KUKA KRL program: EPS_2_25369_MH3A_A_20251215023756.src

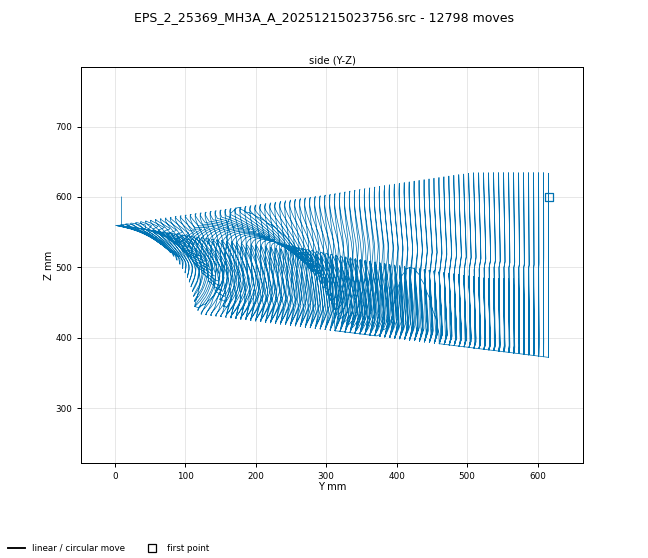
[picture p0: tool path of EPS_2_25369_MH3A_A_20251215023756.src, 12798 of 12800 moves have a stored position in this frame; points joined in program order, loops and branches not executed]
&ACCESS RVP
&REL 4
&COMMENT QRS 19112012
&PARAM EDITMASK = *
DEF PART()
EXT BAS (BAS_COMMAND :IN,REAL :IN )
INT I
BAS (#INITMOV,0 )

;KUKA QRS Post kuka4.cps  Date:22-06-2017 !

File_ID=2956

QRS_PRE_INIT()

;Init var - Until changes are made in qrs_pre_init
Outlet_Square_prg=0
Inlet_1_Square_prg=0
Inlet_2_Square_prg=0
Inlet_3_Square_prg=0
Inlet_4_Square_prg=0
Inlet_5_Square_prg=0

Outlet_1={X 0.000, Y 509.470, Z 509.000, B 0.000, E1 0.000 }
Inlet_1={X 0.000, Y 526.260, Z 384.000, B 0.000, E1 183.000 }
Inlet_2={X 0.000, Y 520.510, Z 359.000, B 0.000, E1 271.000 }
Outlet_1_type=251
Inlet_1_type=201
Inlet_2_type=251
;QRS#1=Sidecore dimensions
;QRS#2=250-10" PVC SDR 35
;QRS#3=200-8" PVC SDR 35
;QRS#4=250-10" PVC SDR 35
;QRS#5=
;QRS#6=
;QRS#7=
;QRS#8=
;QRS#9=14M PSX
;QRS#10=12-08 PSX
;QRS#11=14M PSX
;QRS#12=
;QRS#13=
;QRS#14=
;QRS#15=
;QRS#16=1220x127x914 3'
;QRS#17=EPS Height
;QRS#18=634,5
;QRS#19=*
;QRS#20= UPDATED VERSION 22-06-2017
;QRS#21=*
Outlet_Square=0100
Inlet_1_Square=0100
Inlet_2_Square=0100
Inlet_3_Square=0
Inlet_4_Square=0
Inlet_5_Square=0
Mill_Square=1
Outlet_Square_Prg=205
Inlet_1_Square_prg=204
Inlet_2_Square_prg=205

QRS_INIT()

$ADVANCE=5

; T1
PTP {E1 173.595,E2 173.595}
PTP {X 0,Y 615.506,A -85,B 0,C 180,E1 173.595,E2 173.595,E3 0,E4 0,E5 0,E6 0}
QRS_SPEED_INIT()
LIN {X 0,Y 615.506,Z 600,A -85,B 0,C 180,E1 173.595,E2 173.595,E3 0,E4 0,E5 0,E6 0} C_VEL
LIN {X 0,Y 615.506,Z 382.487,A -85,B 0,C 180,E1 173.595,E2 173.595} C_VEL
LIN {X 0,Y 615.506,Z 374.307,A -85,B 0,C 180,E1 173.595,E2 173.595} C_VEL
LIN {X 0,Y 615.49,Z 372.307,A -85,B 0,C 180,E1 173.408,E2 173.408} C_VEL
LIN {X 0,Y 615.486,Z 372.321,A -85,B 0,C 180,E1 170.801,E2 170.801} C_VEL
LIN {X 0,Y 615.474,Z 372.316,A -85,B 0,C 180,E1 168.139,E2 168.139} C_VEL
LIN {X 0,Y 615.49,Z 372.307,A -85,B 0,C 180,E1 165.451,E2 165.451} C_VEL
LIN {X 0,Y 615.494,Z 372.324,A -85,B 0,C 180,E1 162.729,E2 162.729} C_VEL
LIN {X 0,Y 615.479,Z 372.311,A -85,B 0,C 180,E1 159.967,E2 159.967} C_VEL
LIN {X 0,Y 615.491,Z 372.306,A -85,B 0,C 180,E1 157.65,E2 157.65} C_VEL
LIN {X 0,Y 615.48,Z 372.319,A -85,B 0,C 180,E1 155.008,E2 155.008} C_VEL
LIN {X 0,Y 615.487,Z 372.324,A -85,B 0,C 180,E1 152.822,E2 152.822} C_VEL
LIN {X 0,Y 615.477,Z 372.314,A -85,B 0,C 180,E1 150.205,E2 150.205} C_VEL
LIN {X 0,Y 615.49,Z 372.307,A -85,B 0,C 180,E1 147.542,E2 147.542} C_VEL
LIN {X 0,Y 615.481,Z 372.316,A -85,B 0,C 180,E1 145.184,E2 145.184} C_VEL
LIN {X 0,Y 615.494,Z 372.325,A -85,B 0,C 180,E1 142.758,E2 142.758} C_VEL
LIN {X 0,Y 615.486,Z 372.307,A -85,B 0,C 180,E1 139.909,E2 139.909} C_VEL
LIN {X 0,Y 615.494,Z 372.306,A -85,B 0,C 180,E1 137.647,E2 137.647} C_VEL
LIN {X 0,Y 615.491,Z 372.324,A -85,B 0,C 180,E1 134.931,E2 134.931} C_VEL
LIN {X 0,Y 615.48,Z 372.31,A -85,B 0,C 180,E1 132.079,E2 132.079} C_VEL
LIN {X 0,Y 615.494,Z 372.306,A -85,B 0,C 180,E1 129.748,E2 129.748} C_VEL
LIN {X 0,Y 615.488,Z 372.327,A -85,B 0,C 180,E1 126.936,E2 126.936} C_VEL
LIN {X 0,Y 615.491,Z 372.319,A -85,B 0,C 180,E1 124.7,E2 124.7} C_VEL
LIN {X 0,Y 615.477,Z 372.312,A -85,B 0,C 180,E1 122.328,E2 122.328} C_VEL
LIN {X 0,Y 615.497,Z 372.305,A -85,B 0,C 180,E1 119.795,E2 119.795} C_VEL
LIN {X 0,Y 615.491,Z 372.325,A -85,B 0,C 180,E1 117.045,E2 117.045} C_VEL
LIN {X 0,Y 615.478,Z 372.311,A -85,B 0,C 180,E1 114.271,E2 114.271} C_VEL
LIN {X 0,Y 615.481,Z 372.316,A -85,B 0,C 180,E1 111.431,E2 111.431} C_VEL
LIN {X 0,Y 615.481,Z 372.315,A -85,B 0,C 180,E1 108.602,E2 108.602} C_VEL
LIN {X 0,Y 615.487,Z 372.308,A -85,B 0,C 180,E1 105.904,E2 105.904} C_VEL
LIN {X 0,Y 615.49,Z 372.321,A -85,B 0,C 180,E1 105.225,E2 105.225} C_VEL
LIN {X 0,Y 615.478,Z 375.734,A -85,B 0,C 180,E1 102.529,E2 102.529} C_VEL
LIN {X 0,Y 615.491,Z 379.183,A -85,B 0,C 180,E1 99.861,E2 99.861} C_VEL
LIN {X 0,Y 615.482,Z 380.919,A -85,B 0,C 180,E1 98.536,E2 98.536} C_VEL
LIN {X 0,Y 615.488,Z 393.813,A -85,B 0,C 180,E1 98.246,E2 98.246} C_VEL
LIN {X 0,Y 615.485,Z 406.345,A -85,B 0,C 180,E1 97.834,E2 97.834} C_VEL
LIN {X 0,Y 615.478,Z 418.326,A -85,B 0,C 180,E1 97.297,E2 97.297} C_VEL
LIN {X 0,Y 615.495,Z 429.344,A -85,B 0,C 180,E1 96.661,E2 96.661} C_VEL
LIN {X 0,Y 615.5,Z 439.937,A -85,B 0,C 180,E1 95.898,E2 95.898} C_VEL
LIN {X 0,Y 615.498,Z 449.187,A -85,B 0,C 180,E1 95.076,E2 95.076} C_VEL
LIN {X 0,Y 615.499,Z 458.111,A -85,B 0,C 180,E1 94.092,E2 94.092} C_VEL
LIN {X 0,Y 615.497,Z 465.316,A -85,B 0,C 180,E1 93.108,E2 93.108} C_VEL
LIN {X 0,Y 615.5,Z 471.91,A -85,B 0,C 180,E1 91.962,E2 91.962} C_VEL
LIN {X 0,Y 615.497,Z 476.278,A -85,B 0,C 180,E1 90.981,E2 90.981} C_VEL
LIN {X 0,Y 615.496,Z 479.593,A -85,B 0,C 180,E1 89.999,E2 89.999} C_VEL
LIN {X 0,Y 615.498,Z 482.486,A -85,B 0,C 180,E1 88.691,E2 88.691} C_VEL
LIN {X 0,Y 615.499,Z 483.348,A -85,B 0,C 180,E1 88.036,E2 88.036} C_VEL
LIN {X 0,Y 615.496,Z 483.794,A -85,B 0,C 180,E1 87.381,E2 87.381} C_VEL
LIN {X 0,Y 615.495,Z 483.512,A -85,B 0,C 180,E1 86.071,E2 86.071} C_VEL
LIN {X 0,Y 615.496,Z 482.804,A -85,B 0,C 180,E1 85.415,E2 85.415} C_VEL
LIN {X 0,Y 615.496,Z 481.658,A -85,B 0,C 180,E1 84.758,E2 84.758} C_VEL
LIN {X 0,Y 615.497,Z 480.101,A -85,B 0,C 180,E1 84.101,E2 84.101} C_VEL
LIN {X 0,Y 615.497,Z 476.921,A -85,B 0,C 180,E1 83.101,E2 83.101} C_VEL
LIN {X 0,Y 615.495,Z 472.771,A -85,B 0,C 180,E1 82.124,E2 82.124} C_VEL
LIN {X 0,Y 615.496,Z 466.374,A -85,B 0,C 180,E1 80.966,E2 80.966} C_VEL
LIN {X 0,Y 615.497,Z 459.364,A -85,B 0,C 180,E1 79.971,E2 79.971} C_VEL
LIN {X 0,Y 615.498,Z 450.403,A -85,B 0,C 180,E1 78.958,E2 78.958} C_VEL
LIN {X 0,Y 615.497,Z 441.497,A -85,B 0,C 180,E1 78.139,E2 78.139} C_VEL
LIN {X 0,Y 615.5,Z 431.437,A -85,B 0,C 180,E1 77.386,E2 77.386} C_VEL
LIN {X 0,Y 615.477,Z 420.231,A -85,B 0,C 180,E1 76.714,E2 76.714} C_VEL
LIN {X 0,Y 615.487,Z 409.605,A -85,B 0,C 180,E1 76.209,E2 76.209} C_VEL
LIN {X 0,Y 615.491,Z 397.137,A -85,B 0,C 180,E1 75.758,E2 75.758} C_VEL
LIN {X 0,Y 615.484,Z 383.804,A -85,B 0,C 180,E1 75.429,E2 75.429} C_VEL
LIN {X 0,Y 615.484,Z 380.908,A -85,B 0,C 180,E1 75.366,E2 75.366} C_VEL
LIN {X 0,Y 615.477,Z 377.471,A -85,B 0,C 180,E1 72.729,E2 72.729} C_VEL
LIN {X 0,Y 615.486,Z 373.927,A -85,B 0,C 180,E1 69.967,E2 69.967} C_VEL
LIN {X 0,Y 615.487,Z 372.319,A -85,B 0,C 180,E1 68.568,E2 68.568} C_VEL
LIN {X 0,Y 615.478,Z 372.311,A -85,B 0,C 180,E1 65.727,E2 65.727} C_VEL
LIN {X 0,Y 615.491,Z 372.324,A -85,B 0,C 180,E1 62.955,E2 62.955} C_VEL
LIN {X 0,Y 615.497,Z 372.306,A -85,B 0,C 180,E1 60.205,E2 60.205} C_VEL
LIN {X 0,Y 615.481,Z 372.318,A -85,B 0,C 180,E1 57.542,E2 57.542} C_VEL
LIN {X 0,Y 615.499,Z 372.322,A -85,B 0,C 180,E1 55.185,E2 55.185} C_VEL
LIN {X 0,Y 615.477,Z 372.313,A -85,B 0,C 180,E1 52.757,E2 52.757} C_VEL
LIN {X 0,Y 615.483,Z 372.315,A -85,B 0,C 180,E1 49.912,E2 49.912} C_VEL
LIN {X 0,Y 615.49,Z 372.323,A -85,B 0,C 180,E1 47.647,E2 47.647} C_VEL
LIN {X 0,Y 615.48,Z 372.312,A -85,B 0,C 180,E1 44.93,E2 44.93} C_VEL
LIN {X 0,Y 615.494,Z 372.315,A -85,B 0,C 180,E1 42.08,E2 42.08} C_VEL
LIN {X 0,Y 615.496,Z 372.324,A -85,B 0,C 180,E1 39.75,E2 39.75} C_VEL
LIN {X 0,Y 615.478,Z 372.31,A -85,B 0,C 180,E1 36.935,E2 36.935} C_VEL
LIN {X 0,Y 615.494,Z 372.325,A -85,B 0,C 180,E1 34.022,E2 34.022} C_VEL
LIN {X 0,Y 615.479,Z 372.318,A -85,B 0,C 180,E1 31.686,E2 31.686} C_VEL
LIN {X 0,Y 615.487,Z 372.31,A -85,B 0,C 180,E1 29.407,E2 29.407} C_VEL
LIN {X 0,Y 615.493,Z 372.319,A -85,B 0,C 180,E1 26.444,E2 26.444} C_VEL
LIN {X 0,Y 615.485,Z 372.31,A -85,B 0,C 180,E1 23.557,E2 23.557} C_VEL
LIN {X 0,Y 615.48,Z 372.319,A -85,B 0,C 180,E1 20.731,E2 20.731} C_VEL
LIN {X 0,Y 615.477,Z 372.314,A -85,B 0,C 180,E1 17.957,E2 17.957} C_VEL
LIN {X 0,Y 615.487,Z 372.311,A -85,B 0,C 180,E1 15.226,E2 15.226} C_VEL
LIN {X 0,Y 615.499,Z 372.323,A -85,B 0,C 180,E1 12.635,E2 12.635} C_VEL
LIN {X 0,Y 615.483,Z 386.641,A -85,B 0,C 180,E1 12.196,E2 12.196} C_VEL
LIN {X 0,Y 615.482,Z 398.98,A -85,B 0,C 180,E1 11.694,E2 11.694} C_VEL
LIN {X 0,Y 615.484,Z 411.621,A -85,B 0,C 180,E1 11.041,E2 11.041} C_VEL
LIN {X 0,Y 615.498,Z 423.541,A -85,B 0,C 180,E1 10.278,E2 10.278} C_VEL
LIN {X 0,Y 615.496,Z 435.177,A -85,B 0,C 180,E1 9.365,E2 9.365} C_VEL
LIN {X 0,Y 615.497,Z 445.582,A -85,B 0,C 180,E1 8.371,E2 8.371} C_VEL
LIN {X 0,Y 615.497,Z 454.162,A -85,B 0,C 180,E1 7.381,E2 7.381} C_VEL
LIN {X 0,Y 615.495,Z 462.378,A -85,B 0,C 180,E1 6.228,E2 6.228} C_VEL
LIN {X 0,Y 615.494,Z 468.108,A -85,B 0,C 180,E1 5.241,E2 5.241} C_VEL
LIN {X 0,Y 615.493,Z 472.821,A -85,B 0,C 180,E1 4.257,E2 4.257} C_VEL
LIN {X 0,Y 615.491,Z 477.703,A -85,B 0,C 180,E1 2.946,E2 2.946} C_VEL
LIN {X 0,Y 615.495,Z 480.406,A -85,B 0,C 180,E1 1.963,E2 1.963} C_VEL
LIN {X 0,Y 615.491,Z 482.766,A -85,B 0,C 180,E1 0.654,E2 0.654} C_VEL
LIN {X 0,Y 615.49,Z 483.802,A -85,B 0,C 180,E1 -0.654,E2 -0.654} C_VEL
LIN {X 0,Y 615.495,Z 483.535,A -85,B 0,C 180,E1 -1.963,E2 -1.963} C_VEL
LIN {X 0,Y 615.497,Z 481.964,A -85,B 0,C 180,E1 -3.273,E2 -3.273} C_VEL
LIN {X 0,Y 615.495,Z 479.039,A -85,B 0,C 180,E1 -4.584,E2 -4.584} C_VEL
LIN {X 0,Y 615.49,Z 474.68,A -85,B 0,C 180,E1 -5.898,E2 -5.898} C_VEL
LIN {X 0,Y 615.495,Z 470.285,A -85,B 0,C 180,E1 -6.899,E2 -6.899} C_VEL
LIN {X 0,Y 615.497,Z 464.066,A -85,B 0,C 180,E1 -8.041,E2 -8.041} C_VEL
LIN {X 0,Y 615.498,Z 456.232,A -85,B 0,C 180,E1 -9.198,E2 -9.198} C_VEL
LIN {X 0,Y 615.496,Z 448.03,A -85,B 0,C 180,E1 -10.194,E2 -10.194} C_VEL
LIN {X 0,Y 615.496,Z 438.135,A -85,B 0,C 180,E1 -11.193,E2 -11.193} C_VEL
LIN {X 0,Y 615.498,Z 427.094,A -85,B 0,C 180,E1 -12.111,E2 -12.111} C_VEL
LIN {X 0,Y 615.495,Z 414.683,A -85,B 0,C 180,E1 -12.949,E2 -12.949} C_VEL
LIN {X 0,Y 615.491,Z 402.363,A -85,B 0,C 180,E1 -13.621,E2 -13.621} C_VEL
LIN {X 0,Y 615.497,Z 388.866,A -85,B 0,C 180,E1 -14.202,E2 -14.202} C_VEL
LIN {X 0,Y 615.485,Z 375.572,A -85,B 0,C 180,E1 -14.634,E2 -14.634} C_VEL
LIN {X 0,Y 615.48,Z 372.321,A -85,B 0,C 180,E1 -14.739,E2 -14.739} C_VEL
LIN {X 0,Y 615.492,Z 372.319,A -85,B 0,C 180,E1 -17.27,E2 -17.27} C_VEL
LIN {X 0,Y 615.482,Z 372.323,A -85,B 0,C 180,E1 -20.033,E2 -20.033} C_VEL
LIN {X 0,Y 615.493,Z 372.326,A -85,B 0,C 180,E1 -22.844,E2 -22.844} C_VEL
LIN {X 0,Y 615.484,Z 372.324,A -85,B 0,C 180,E1 -25.568,E2 -25.568} C_VEL
LIN {X 0,Y 615.491,Z 372.319,A -85,B 0,C 180,E1 -28.451,E2 -28.451} C_VEL
LIN {X 0,Y 615.483,Z 372.321,A -85,B 0,C 180,E1 -31.085,E2 -31.085} C_VEL
LIN {X 0,Y 615.489,Z 372.319,A -85,B 0,C 180,E1 -33.534,E2 -33.534} C_VEL
LIN {X 0,Y 615.494,Z 372.323,A -85,B 0,C 180,E1 -36.424,E2 -36.424} C_VEL
LIN {X 0,Y 615.495,Z 372.326,A -85,B 0,C 180,E1 -39.063,E2 -39.063} C_VEL
LIN {X 0,Y 615.496,Z 372.324,A -85,B 0,C 180,E1 -41.473,E2 -41.473} C_VEL
LIN {X 0,Y 615.499,Z 372.323,A -85,B 0,C 180,E1 -44.149,E2 -44.149} C_VEL
LIN {X 0,Y 615.489,Z 372.32,A -85,B 0,C 180,E1 -46.952,E2 -46.952} C_VEL
LIN {X 0,Y 615.484,Z 372.322,A -85,B 0,C 180,E1 -49.393,E2 -49.393} C_VEL
LIN {X 0,Y 615.498,Z 372.377,A -85,B 0,C 180,E1 -52.231,E2 -52.231} C_VEL
LIN {X 0,Y 615.495,Z 388.356,A -85,B 0,C 180,E1 -54.986,E2 -54.986} C_VEL
LIN {X 0,Y 615.483,Z 393.853,A -85,B 0,C 180,E1 -55.977,E2 -55.977} C_VEL
LIN {X 0,Y 615.476,Z 406.828,A -85,B 0,C 180,E1 -58.615,E2 -58.615} C_VEL
LIN {X 0,Y 615.488,Z 420.627,A -85,B 0,C 180,E1 -61.342,E2 -61.342} C_VEL
LIN {X 0,Y 615.484,Z 434.012,A -85,B 0,C 180,E1 -63.92,E2 -63.92} C_VEL
LIN {X 0,Y 615.48,Z 447.386,A -85,B 0,C 180,E1 -66.443,E2 -66.443} C_VEL
LIN {X 0,Y 615.49,Z 462.656,A -85,B 0,C 180,E1 -69.269,E2 -69.269} C_VEL
LIN {X 0,Y 615.495,Z 477.912,A -85,B 0,C 180,E1 -72.043,E2 -72.043} C_VEL
LIN {X 0,Y 615.48,Z 493.156,A -85,B 0,C 180,E1 -74.773,E2 -74.773} C_VEL
LIN {X 0,Y 615.489,Z 499.56,A -85,B 0,C 180,E1 -75.911,E2 -75.911} C_VEL
LIN {X 0,Y 615.49,Z 515.549,A -85,B 0,C 180,E1 -76.167,E2 -76.167} C_VEL
LIN {X 0,Y 615.48,Z 528.9,A -85,B 0,C 180,E1 -76.504,E2 -76.504} C_VEL
LIN {X 0,Y 615.497,Z 542.13,A -85,B 0,C 180,E1 -76.966,E2 -76.966} C_VEL
LIN {X 0,Y 615.478,Z 555.006,A -85,B 0,C 180,E1 -77.553,E2 -77.553} C_VEL
LIN {X 0,Y 615.497,Z 566.763,A -85,B 0,C 180,E1 -78.222,E2 -78.222} C_VEL
LIN {X 0,Y 615.496,Z 577.409,A -85,B 0,C 180,E1 -78.957,E2 -78.957} C_VEL
LIN {X 0,Y 615.498,Z 587.635,A -85,B 0,C 180,E1 -79.805,E2 -79.805} C_VEL
LIN {X 0,Y 615.498,Z 597.582,A -85,B 0,C 180,E1 -80.801,E2 -80.801} C_VEL
LIN {X 0,Y 615.496,Z 607.068,A -85,B 0,C 180,E1 -81.959,E2 -81.959} C_VEL
LIN {X 0,Y 615.495,Z 614.651,A -85,B 0,C 180,E1 -83.1,E2 -83.1} C_VEL
LIN {X 0,Y 615.494,Z 620.067,A -85,B 0,C 180,E1 -84.101,E2 -84.101} C_VEL
LIN {X 0,Y 615.495,Z 625.68,A -85,B 0,C 180,E1 -85.415,E2 -85.415} C_VEL
LIN {X 0,Y 615.495,Z 629.752,A -85,B 0,C 180,E1 -86.726,E2 -86.726} C_VEL
LIN {X 0,Y 615.498,Z 632.405,A -85,B 0,C 180,E1 -88.036,E2 -88.036} C_VEL
LIN {X 0,Y 615.493,Z 633.722,A -85,B 0,C 180,E1 -89.345,E2 -89.345} C_VEL
LIN {X 0,Y 615.493,Z 633.723,A -85,B 0,C 180,E1 -90.654,E2 -90.654} C_VEL
LIN {X 0,Y 615.497,Z 632.407,A -85,B 0,C 180,E1 -91.962,E2 -91.962} C_VEL
LIN {X 0,Y 615.495,Z 629.756,A -85,B 0,C 180,E1 -93.272,E2 -93.272} C_VEL
LIN {X 0,Y 615.495,Z 625.686,A -85,B 0,C 180,E1 -94.584,E2 -94.584} C_VEL
LIN {X 0,Y 615.494,Z 620.074,A -85,B 0,C 180,E1 -95.898,E2 -95.898} C_VEL
LIN {X 0,Y 615.495,Z 614.656,A -85,B 0,C 180,E1 -96.899,E2 -96.899} C_VEL
LIN {X 0,Y 615.496,Z 607.078,A -85,B 0,C 180,E1 -98.04,E2 -98.04} C_VEL
LIN {X 0,Y 615.498,Z 597.594,A -85,B 0,C 180,E1 -99.198,E2 -99.198} C_VEL
LIN {X 0,Y 615.498,Z 587.65,A -85,B 0,C 180,E1 -100.193,E2 -100.193} C_VEL
LIN {X 0,Y 615.498,Z 576.393,A -85,B 0,C 180,E1 -101.117,E2 -101.117} C_VEL
LIN {X 0,Y 615.496,Z 565.429,A -85,B 0,C 180,E1 -101.86,E2 -101.86} C_VEL
LIN {X 0,Y 615.479,Z 553.347,A -85,B 0,C 180,E1 -102.529,E2 -102.529} C_VEL
LIN {X 0,Y 615.496,Z 539.952,A -85,B 0,C 180,E1 -103.116,E2 -103.116} C_VEL
LIN {X 0,Y 615.479,Z 525.927,A -85,B 0,C 180,E1 -103.579,E2 -103.579} C_VEL
LIN {X 0,Y 615.495,Z 511.649,A -85,B 0,C 180,E1 -103.905,E2 -103.905} C_VEL
LIN {X 0,Y 615.489,Z 499.562,A -85,B 0,C 180,E1 -104.089,E2 -104.089} C_VEL
LIN {X 0,Y 615.494,Z 483.64,A -85,B 0,C 180,E1 -106.927,E2 -106.927} C_VEL
LIN {X 0,Y 615.485,Z 468.39,A -85,B 0,C 180,E1 -109.684,E2 -109.684} C_VEL
LIN {X 0,Y 615.477,Z 453.911,A -85,B 0,C 180,E1 -112.343,E2 -112.343} C_VEL
LIN {X 0,Y 615.493,Z 439.753,A -85,B 0,C 180,E1 -114.99,E2 -114.99} C_VEL
LIN {X 0,Y 615.481,Z 426.373,A -85,B 0,C 180,E1 -117.545,E2 -117.545} C_VEL
LIN {X 0,Y 615.478,Z 412.986,A -85,B 0,C 180,E1 -120.159,E2 -120.159} C_VEL
LIN {X 0,Y 615.49,Z 399.598,A -85,B 0,C 180,E1 -122.845,E2 -122.845} C_VEL
LIN {X 0,Y 615.487,Z 386.802,A -85,B 0,C 180,E1 -125.414,E2 -125.414} C_VEL
LIN {X 0,Y 615.482,Z 373.652,A -85,B 0,C 180,E1 -128.068,E2 -128.068} C_VEL
LIN {X 0,Y 615.478,Z 372.314,A -85,B 0,C 180,E1 -128.38,E2 -128.38} C_VEL
LIN {X 0,Y 615.48,Z 372.31,A -85,B 0,C 180,E1 -131.094,E2 -131.094} C_VEL
LIN {X 0,Y 615.484,Z 372.321,A -85,B 0,C 180,E1 -133.997,E2 -133.997} C_VEL
LIN {X 0,Y 615.498,Z 372.305,A -85,B 0,C 180,E1 -136.756,E2 -136.756} C_VEL
LIN {X 0,Y 615.479,Z 372.317,A -85,B 0,C 180,E1 -139.393,E2 -139.393} C_VEL
LIN {X 0,Y 615.484,Z 372.32,A -85,B 0,C 180,E1 -141.987,E2 -141.987} C_VEL
LIN {X 0,Y 615.481,Z 372.311,A -85,B 0,C 180,E1 -144.384,E2 -144.384} C_VEL
LIN {X 0,Y 615.488,Z 372.307,A -85,B 0,C 180,E1 -146.764,E2 -146.764} C_VEL
LIN {X 0,Y 615.478,Z 372.312,A -85,B 0,C 180,E1 -149.08,E2 -149.08} C_VEL
LIN {X 0,Y 615.491,Z 372.322,A -85,B 0,C 180,E1 -151.546,E2 -151.546} C_VEL
LIN {X 0,Y 615.485,Z 372.309,A -85,B 0,C 180,E1 -154.429,E2 -154.429} C_VEL
LIN {X 0,Y 615.475,Z 372.316,A -85,B 0,C 180,E1 -157.155,E2 -157.155} C_VEL
LIN {X 0,Y 615.487,Z 372.321,A -85,B 0,C 180,E1 -159.44,E2 -159.44} C_VEL
LIN {X 0,Y 615.477,Z 372.316,A -85,B 0,C 180,E1 -162.043,E2 -162.043} C_VEL
LIN {X 0,Y 615.486,Z 372.308,A -85,B 0,C 180,E1 -164.774,E2 -164.774} C_VEL
LIN {X 0,Y 615.485,Z 372.325,A -85,B 0,C 180,E1 -167.47,E2 -167.47} C_VEL
LIN {X 0,Y 615.477,Z 372.313,A -85,B 0,C 180,E1 -170.138,E2 -170.138} C_VEL
LIN {X 0,Y 615.483,Z 372.309,A -85,B 0,C 180,E1 -172.784,E2 -172.784} C_VEL
LIN {X 0,Y 615.493,Z 372.323,A -85,B 0,C 180,E1 -175.416,E2 -175.416} C_VEL
LIN {X 0,Y 615.477,Z 372.314,A -85,B 0,C 180,E1 -178.037,E2 -178.037} C_VEL
LIN {X 0,Y 615.486,Z 372.308,A -85,B 0,C 180,E1 -180.654,E2 -180.654} C_VEL
LIN {X 0,Y 615.486,Z 372.322,A -85,B 0,C 180,E1 -183.273,E2 -183.273} C_VEL
LIN {X 0,Y 615.476,Z 372.316,A -85,B 0,C 180,E1 -185.899,E2 -185.899} C_VEL
LIN {X 0,Y 615.49,Z 372.307,A -85,B 0,C 180,E1 -186.592,E2 -186.592} C_VEL
LIN {X 0,Y 614.81,Z 372.468,A -85,B 0,C 180,E1 -187.138,E2 -187.138} C_VEL
LIN {X 0,Y 611.974,Z 372.875,A -85,B 0,C 180,E1 -188.024,E2 -188.024} C_VEL
LIN {X 0,Y 609.582,Z 373.191,A -85,B 0,C 180,E1 -188.736,E2 -188.736} C_VEL
LIN {X 0,Y 608.545,Z 373.31,A -85,B 0,C 180,E1 -189.286,E2 -189.286} C_VEL
LIN {X 0,Y 608.455,Z 373.318,A -85,B 0,C 180,E1 -189.472,E2 -189.472} C_VEL
LIN {X 0,Y 608.452,Z 373.314,A -85,B 0,C 180,E1 -192,E2 -192} C_VEL
LIN {X 0,Y 608.476,Z 373.311,A -85,B 0,C 180,E1 -194.721,E2 -194.721} C_VEL
LIN {X 0,Y 608.454,Z 373.32,A -85,B 0,C 180,E1 -197.477,E2 -197.477} C_VEL
LIN {X 0,Y 608.459,Z 373.311,A -85,B 0,C 180,E1 -200.275,E2 -200.275} C_VEL
LIN {X 0,Y 608.455,Z 373.312,A -85,B 0,C 180,E1 -202.479,E2 -202.479} C_VEL
LIN {X 0,Y 608.451,Z 373.313,A -85,B 0,C 180,E1 -204.571,E2 -204.571} C_VEL
LIN {X 0,Y 608.478,Z 373.319,A -85,B 0,C 180,E1 -207.21,E2 -207.21} C_VEL
LIN {X 0,Y 608.461,Z 373.312,A -85,B 0,C 180,E1 -209.973,E2 -209.973} C_VEL
LIN {X 0,Y 608.463,Z 373.312,A -85,B 0,C 180,E1 -212.525,E2 -212.525} C_VEL
LIN {X 0,Y 608.439,Z 373.324,A -85,B 0,C 180,E1 -215.278,E2 -215.278} C_VEL
LIN {X 0,Y 608.468,Z 373.313,A -85,B 0,C 180,E1 -217.747,E2 -217.747} C_VEL
LIN {X 0,Y 608.45,Z 373.313,A -85,B 0,C 180,E1 -220.331,E2 -220.331} C_VEL
LIN {X 0,Y 608.484,Z 373.316,A -85,B 0,C 180,E1 -223.312,E2 -223.312} C_VEL
LIN {X 0,Y 608.468,Z 373.31,A -85,B 0,C 180,E1 -226.132,E2 -226.132} C_VEL
LIN {X 0,Y 608.456,Z 373.318,A -85,B 0,C 180,E1 -228.825,E2 -228.825} C_VEL
LIN {X 0,Y 608.472,Z 373.315,A -85,B 0,C 180,E1 -231.414,E2 -231.414} C_VEL
LIN {X 0,Y 608.476,Z 373.31,A -85,B 0,C 180,E1 -233.951,E2 -233.951} C_VEL
LIN {X 0,Y 608.462,Z 373.312,A -85,B 0,C 180,E1 -236.33,E2 -236.33} C_VEL
LIN {X 0,Y 608.477,Z 373.315,A -85,B 0,C 180,E1 -238.729,E2 -238.729} C_VEL
LIN {X 0,Y 608.469,Z 373.315,A -85,B 0,C 180,E1 -241.382,E2 -241.382} C_VEL
LIN {X 0,Y 608.445,Z 373.313,A -85,B 0,C 180,E1 -243.966,E2 -243.966} C_VEL
LIN {X 0,Y 608.464,Z 373.311,A -85,B 0,C 180,E1 -246.156,E2 -246.156} C_VEL
LIN {X 0,Y 608.456,Z 373.322,A -85,B 0,C 180,E1 -249.02,E2 -249.02} C_VEL
LIN {X 0,Y 608.454,Z 373.312,A -85,B 0,C 180,E1 -251.829,E2 -251.829} C_VEL
LIN {X 0,Y 608.474,Z 373.315,A -85,B 0,C 180,E1 -254.595,E2 -254.595} C_VEL
LIN {X 0,Y 608.408,Z 373.638,A -85,B 0,C 180,E1 -255.279,E2 -255.279} C_VEL
LIN {X 0,Y 608.436,Z 377.105,A -85,B 0,C 180,E1 -258.001,E2 -258.001} C_VEL
LIN {X 0,Y 608.409,Z 380.582,A -85,B 0,C 180,E1 -260.694,E2 -260.694} C_VEL
LIN {X 0,Y 608.414,Z 381.398,A -85,B 0,C 180,E1 -261.322,E2 -261.322} C_VEL
LIN {X 0,Y 608.539,Z 396.686,A -85,B 0,C 180,E1 -261.7,E2 -261.7} C_VEL
LIN {X 0,Y 608.506,Z 408.414,A -85,B 0,C 180,E1 -262.118,E2 -262.118} C_VEL
LIN {X 0,Y 608.496,Z 420.708,A -85,B 0,C 180,E1 -262.702,E2 -262.702} C_VEL
LIN {X 0,Y 608.483,Z 431.71,A -85,B 0,C 180,E1 -263.368,E2 -263.368} C_VEL
LIN {X 0,Y 608.498,Z 440.641,A -85,B 0,C 180,E1 -264.034,E2 -264.034} C_VEL
LIN {X 0,Y 608.483,Z 449.843,A -85,B 0,C 180,E1 -264.865,E2 -264.865} C_VEL
LIN {X 0,Y 608.474,Z 458.772,A -85,B 0,C 180,E1 -265.861,E2 -265.861} C_VEL
LIN {X 0,Y 608.458,Z 465.982,A -85,B 0,C 180,E1 -266.856,E2 -266.856} C_VEL
LIN {X 0,Y 608.445,Z 472.572,A -85,B 0,C 180,E1 -268.015,E2 -268.015} C_VEL
LIN {X 0,Y 608.428,Z 476.942,A -85,B 0,C 180,E1 -269.008,E2 -269.008} C_VEL
LIN {X 0,Y 608.436,Z 480.253,A -85,B 0,C 180,E1 -270.001,E2 -270.001} C_VEL
LIN {X 0,Y 608.45,Z 483.142,A -85,B 0,C 180,E1 -271.324,E2 -271.324} C_VEL
LIN {X 0,Y 608.444,Z 483.993,A -85,B 0,C 180,E1 -271.987,E2 -271.987} C_VEL
LIN {X 0,Y 608.422,Z 484.444,A -85,B 0,C 180,E1 -273.312,E2 -273.312} C_VEL
LIN {X 0,Y 608.432,Z 484.095,A -85,B 0,C 180,E1 -273.975,E2 -273.975} C_VEL
LIN {X 0,Y 608.429,Z 483.351,A -85,B 0,C 180,E1 -274.639,E2 -274.639} C_VEL
LIN {X 0,Y 608.438,Z 482.168,A -85,B 0,C 180,E1 -275.303,E2 -275.303} C_VEL
LIN {X 0,Y 608.448,Z 478.667,A -85,B 0,C 180,E1 -276.603,E2 -276.603} C_VEL
LIN {X 0,Y 608.449,Z 474.659,A -85,B 0,C 180,E1 -277.634,E2 -277.634} C_VEL
LIN {X 0,Y 608.451,Z 469.6,A -85,B 0,C 180,E1 -278.637,E2 -278.637} C_VEL
LIN {X 0,Y 608.467,Z 463.229,A -85,B 0,C 180,E1 -279.642,E2 -279.642} C_VEL
LIN {X 0,Y 608.451,Z 455.224,A -85,B 0,C 180,E1 -280.651,E2 -280.651} C_VEL
LIN {X 0,Y 608.471,Z 447.052,A -85,B 0,C 180,E1 -281.493,E2 -281.493} C_VEL
LIN {X 0,Y 608.477,Z 437.062,A -85,B 0,C 180,E1 -282.339,E2 -282.339} C_VEL
LIN {X 0,Y 608.499,Z 425.741,A -85,B 0,C 180,E1 -283.101,E2 -283.101} C_VEL
LIN {X 0,Y 608.503,Z 414.627,A -85,B 0,C 180,E1 -283.696,E2 -283.696} C_VEL
LIN {X 0,Y 608.534,Z 402.268,A -85,B 0,C 180,E1 -284.207,E2 -284.207} C_VEL
LIN {X 0,Y 608.541,Z 389.139,A -85,B 0,C 180,E1 -284.591,E2 -284.591} C_VEL
LIN {X 0,Y 608.438,Z 381.401,A -85,B 0,C 180,E1 -284.765,E2 -284.765} C_VEL
LIN {X 0,Y 608.407,Z 377.891,A -85,B 0,C 180,E1 -287.478,E2 -287.478} C_VEL
LIN {X 0,Y 608.426,Z 374.316,A -85,B 0,C 180,E1 -290.276,E2 -290.276} C_VEL
LIN {X 0,Y 608.42,Z 373.42,A -85,B 0,C 180,E1 -290.983,E2 -290.983} C_VEL
LIN {X 0,Y 608.454,Z 373.323,A -85,B 0,C 180,E1 -293.124,E2 -293.124} C_VEL
LIN {X 0,Y 608.475,Z 373.311,A -85,B 0,C 180,E1 -295.721,E2 -295.721} C_VEL
LIN {X 0,Y 608.446,Z 373.315,A -85,B 0,C 180,E1 -298.267,E2 -298.267} C_VEL
LIN {X 0,Y 608.471,Z 373.316,A -85,B 0,C 180,E1 -300.545,E2 -300.545} C_VEL
LIN {X 0,Y 608.453,Z 373.321,A -85,B 0,C 180,E1 -302.88,E2 -302.88} C_VEL
LIN {X 0,Y 608.446,Z 373.315,A -85,B 0,C 180,E1 -305.278,E2 -305.278} C_VEL
LIN {X 0,Y 608.468,Z 373.311,A -85,B 0,C 180,E1 -307.747,E2 -307.747} C_VEL
LIN {X 0,Y 608.454,Z 373.319,A -85,B 0,C 180,E1 -310.329,E2 -310.329} C_VEL
LIN {X 0,Y 608.449,Z 373.316,A -85,B 0,C 180,E1 -312.961,E2 -312.961} C_VEL
LIN {X 0,Y 608.463,Z 373.313,A -85,B 0,C 180,E1 -315.736,E2 -315.736} C_VEL
LIN {X 0,Y 608.466,Z 373.315,A -85,B 0,C 180,E1 -318.658,E2 -318.658} C_VEL
LIN {X 0,Y 608.468,Z 373.311,A -85,B 0,C 180,E1 -321.412,E2 -321.412} C_VEL
LIN {X 0,Y 608.482,Z 373.317,A -85,B 0,C 180,E1 -323.95,E2 -323.95} C_VEL
LIN {X 0,Y 608.453,Z 373.317,A -85,B 0,C 180,E1 -326.328,E2 -326.328} C_VEL
LIN {X 0,Y 608.449,Z 373.313,A -85,B 0,C 180,E1 -328.732,E2 -328.732} C_VEL
LIN {X 0,Y 608.473,Z 373.313,A -85,B 0,C 180,E1 -331.38,E2 -331.38} C_VEL
LIN {X 0,Y 608.445,Z 373.32,A -85,B 0,C 180,E1 -333.964,E2 -333.964} C_VEL
LIN {X 0,Y 608.461,Z 373.315,A -85,B 0,C 180,E1 -336.155,E2 -336.155} C_VEL
LIN {X 0,Y 608.472,Z 373.311,A -85,B 0,C 180,E1 -338.308,E2 -338.308} C_VEL
LIN {X 0,Y 608.473,Z 373.317,A -85,B 0,C 180,E1 -341.284,E2 -341.284} C_VEL
LIN {X 0,Y 608.457,Z 373.315,A -85,B 0,C 180,E1 -343.906,E2 -343.906} C_VEL
LIN {X 0,Y 608.46,Z 373.313,A -85,B 0,C 180,E1 -346.643,E2 -346.643} C_VEL
LIN {X 0,Y 608.505,Z 373.481,A -85,B 0,C 180,E1 -347.239,E2 -347.239} C_VEL
LIN {X 0,Y 608.564,Z 386.978,A -85,B 0,C 180,E1 -347.664,E2 -347.664} C_VEL
LIN {X 0,Y 608.548,Z 399.28,A -85,B 0,C 180,E1 -348.171,E2 -348.171} C_VEL
LIN {X 0,Y 608.527,Z 412.603,A -85,B 0,C 180,E1 -348.873,E2 -348.873} C_VEL
LIN {X 0,Y 608.499,Z 424.995,A -85,B 0,C 180,E1 -349.687,E2 -349.687} C_VEL
LIN {X 0,Y 608.48,Z 435.499,A -85,B 0,C 180,E1 -350.526,E2 -350.526} C_VEL
LIN {X 0,Y 608.486,Z 445.941,A -85,B 0,C 180,E1 -351.531,E2 -351.531} C_VEL
LIN {X 0,Y 608.47,Z 454.568,A -85,B 0,C 180,E1 -352.534,E2 -352.534} C_VEL
LIN {X 0,Y 608.45,Z 462.834,A -85,B 0,C 180,E1 -353.7,E2 -353.7} C_VEL
LIN {X 0,Y 608.459,Z 468.608,A -85,B 0,C 180,E1 -354.698,E2 -354.698} C_VEL
LIN {X 0,Y 608.439,Z 473.358,A -85,B 0,C 180,E1 -355.694,E2 -355.694} C_VEL
LIN {X 0,Y 608.446,Z 478.279,A -85,B 0,C 180,E1 -357.02,E2 -357.02} C_VEL
LIN {X 0,Y 608.44,Z 481.004,A -85,B 0,C 180,E1 -358.014,E2 -358.014} C_VEL
LIN {X 0,Y 608.434,Z 483.38,A -85,B 0,C 180,E1 -359.338,E2 -359.338} C_VEL
LIN {X 0,Y 608.433,Z 484.416,A -85,B 0,C 180,E1 -360.662,E2 -360.662} C_VEL
LIN {X 0,Y 608.44,Z 484.135,A -85,B 0,C 180,E1 -361.986,E2 -361.986} C_VEL
LIN {X 0,Y 608.425,Z 482.533,A -85,B 0,C 180,E1 -363.311,E2 -363.311} C_VEL
LIN {X 0,Y 608.428,Z 479.563,A -85,B 0,C 180,E1 -364.638,E2 -364.638} C_VEL
LIN {X 0,Y 608.431,Z 475.141,A -85,B 0,C 180,E1 -365.967,E2 -365.967} C_VEL
LIN {X 0,Y 608.441,Z 470.75,A -85,B 0,C 180,E1 -366.966,E2 -366.966} C_VEL
LIN {X 0,Y 608.462,Z 464.386,A -85,B 0,C 180,E1 -368.134,E2 -368.134} C_VEL
LIN {X 0,Y 608.449,Z 456.468,A -85,B 0,C 180,E1 -369.306,E2 -369.306} C_VEL
LIN {X 0,Y 608.459,Z 448.185,A -85,B 0,C 180,E1 -370.313,E2 -370.313} C_VEL
LIN {X 0,Y 608.491,Z 438.205,A -85,B 0,C 180,E1 -371.323,E2 -371.323} C_VEL
LIN {X 0,Y 608.506,Z 427.059,A -85,B 0,C 180,E1 -372.253,E2 -372.253} C_VEL
LIN {X 0,Y 608.528,Z 414.562,A -85,B 0,C 180,E1 -373.1,E2 -373.1} C_VEL
LIN {X 0,Y 608.549,Z 402.152,A -85,B 0,C 180,E1 -373.78,E2 -373.78} C_VEL
LIN {X 0,Y 608.576,Z 389.199,A -85,B 0,C 180,E1 -374.342,E2 -374.342} C_VEL
LIN {X 0,Y 608.59,Z 375.132,A -85,B 0,C 180,E1 -374.803,E2 -374.803} C_VEL
LIN {X 0,Y 608.464,Z 373.318,A -85,B 0,C 180,E1 -374.87,E2 -374.87} C_VEL
LIN {X 0,Y 608.459,Z 373.319,A -85,B 0,C 180,E1 -377.476,E2 -377.476} C_VEL
LIN {X 0,Y 608.461,Z 373.322,A -85,B 0,C 180,E1 -380.274,E2 -380.274} C_VEL
LIN {X 0,Y 608.461,Z 373.319,A -85,B 0,C 180,E1 -382.476,E2 -382.476} C_VEL
LIN {X 0,Y 608.455,Z 373.319,A -85,B 0,C 180,E1 -384.571,E2 -384.571} C_VEL
LIN {X 0,Y 608.479,Z 373.316,A -85,B 0,C 180,E1 -387.207,E2 -387.207} C_VEL
LIN {X 0,Y 608.463,Z 373.319,A -85,B 0,C 180,E1 -389.97,E2 -389.97} C_VEL
LIN {X 0,Y 608.464,Z 373.321,A -85,B 0,C 180,E1 -392.879,E2 -392.879} C_VEL
LIN {X 0,Y 608.437,Z 373.325,A -85,B 0,C 180,E1 -395.278,E2 -395.278} C_VEL
LIN {X 0,Y 608.476,Z 373.32,A -85,B 0,C 180,E1 -397.746,E2 -397.746} C_VEL
LIN {X 0,Y 608.449,Z 373.324,A -85,B 0,C 180,E1 -400.328,E2 -400.328} C_VEL
LIN {X 0,Y 608.485,Z 373.315,A -85,B 0,C 180,E1 -403.31,E2 -403.31} C_VEL
LIN {X 0,Y 608.47,Z 373.317,A -85,B 0,C 180,E1 -406.13,E2 -406.13} C_VEL
LIN {X 0,Y 608.454,Z 373.321,A -85,B 0,C 180,E1 -408.823,E2 -408.823} C_VEL
LIN {X 0,Y 608.47,Z 373.32,A -85,B 0,C 180,E1 -411.412,E2 -411.412} C_VEL
LIN {X 0,Y 608.494,Z 373.417,A -85,B 0,C 180,E1 -412.163,E2 -412.163} C_VEL
LIN {X 0,Y 608.502,Z 389.342,A -85,B 0,C 180,E1 -414.94,E2 -414.94} C_VEL
LIN {X 0,Y 608.657,Z 399.584,A -85,B 0,C 180,E1 -416.737,E2 -416.737} C_VEL
LIN {X 0,Y 608.61,Z 412.977,A -85,B 0,C 180,E1 -419.463,E2 -419.463} C_VEL
LIN {X 0,Y 608.574,Z 426.365,A -85,B 0,C 180,E1 -422.114,E2 -422.114} C_VEL
LIN {X 0,Y 608.563,Z 439.752,A -85,B 0,C 180,E1 -424.704,E2 -424.704} C_VEL
LIN {X 0,Y 608.518,Z 455.052,A -85,B 0,C 180,E1 -427.596,E2 -427.596} C_VEL
LIN {X 0,Y 608.495,Z 470.352,A -85,B 0,C 180,E1 -430.43,E2 -430.43} C_VEL
LIN {X 0,Y 608.483,Z 485.651,A -85,B 0,C 180,E1 -433.216,E2 -433.216} C_VEL
LIN {X 0,Y 608.484,Z 499.979,A -85,B 0,C 180,E1 -435.761,E2 -435.761} C_VEL
LIN {X 0,Y 608.605,Z 515.549,A -85,B 0,C 180,E1 -436.008,E2 -436.008} C_VEL
LIN {X 0,Y 608.585,Z 528.908,A -85,B 0,C 180,E1 -436.348,E2 -436.348} C_VEL
LIN {X 0,Y 608.563,Z 542.157,A -85,B 0,C 180,E1 -436.815,E2 -436.815} C_VEL
LIN {X 0,Y 608.517,Z 555.061,A -85,B 0,C 180,E1 -437.408,E2 -437.408} C_VEL
LIN {X 0,Y 608.534,Z 568.138,A -85,B 0,C 180,E1 -438.17,E2 -438.17} C_VEL
LIN {X 0,Y 608.507,Z 580.039,A -85,B 0,C 180,E1 -439.027,E2 -439.027} C_VEL
LIN {X 0,Y 608.472,Z 591.384,A -85,B 0,C 180,E1 -440.022,E2 -440.022} C_VEL
LIN {X 0,Y 608.473,Z 600.817,A -85,B 0,C 180,E1 -441.029,E2 -441.029} C_VEL
LIN {X 0,Y 608.453,Z 609.793,A -85,B 0,C 180,E1 -442.199,E2 -442.199} C_VEL
LIN {X 0,Y 608.442,Z 617.224,A -85,B 0,C 180,E1 -443.399,E2 -443.399} C_VEL
LIN {X 0,Y 608.44,Z 623.565,A -85,B 0,C 180,E1 -444.697,E2 -444.697} C_VEL
LIN {X 0,Y 608.431,Z 628.439,A -85,B 0,C 180,E1 -446.025,E2 -446.025} C_VEL
LIN {X 0,Y 608.424,Z 631.83,A -85,B 0,C 180,E1 -447.351,E2 -447.351} C_VEL
LIN {X 0,Y 608.442,Z 633.83,A -85,B 0,C 180,E1 -448.676,E2 -448.676} C_VEL
LIN {X 0,Y 608.433,Z 634.5,A -85,B 0,C 180,E1 -449.999,E2 -449.999} C_VEL
LIN {X 0,Y 608.442,Z 633.831,A -85,B 0,C 180,E1 -451.323,E2 -451.323} C_VEL
LIN {X 0,Y 608.424,Z 631.833,A -85,B 0,C 180,E1 -452.648,E2 -452.648} C_VEL
LIN {X 0,Y 608.431,Z 628.444,A -85,B 0,C 180,E1 -453.973,E2 -453.973} C_VEL
LIN {X 0,Y 608.44,Z 623.571,A -85,B 0,C 180,E1 -455.301,E2 -455.301} C_VEL
LIN {X 0,Y 608.444,Z 617.215,A -85,B 0,C 180,E1 -456.603,E2 -456.603} C_VEL
LIN {X 0,Y 608.453,Z 609.803,A -85,B 0,C 180,E1 -457.799,E2 -457.799} C_VEL
LIN {X 0,Y 608.472,Z 600.83,A -85,B 0,C 180,E1 -458.97,E2 -458.97} C_VEL
LIN {X 0,Y 608.472,Z 591.399,A -85,B 0,C 180,E1 -459.976,E2 -459.976} C_VEL
LIN {X 0,Y 608.505,Z 580.051,A -85,B 0,C 180,E1 -460.973,E2 -460.973} C_VEL
LIN {X 0,Y 608.534,Z 568.16,A -85,B 0,C 180,E1 -461.828,E2 -461.828} C_VEL
LIN {X 0,Y 608.517,Z 555.088,A -85,B 0,C 180,E1 -462.59,E2 -462.59} C_VEL
LIN {X 0,Y 608.563,Z 542.193,A -85,B 0,C 180,E1 -463.183,E2 -463.183} C_VEL
LIN {X 0,Y 608.583,Z 528.212,A -85,B 0,C 180,E1 -463.672,E2 -463.672} C_VEL
LIN {X 0,Y 608.62,Z 514.499,A -85,B 0,C 180,E1 -464.012,E2 -464.012} C_VEL
LIN {X 0,Y 608.462,Z 499.771,A -85,B 0,C 180,E1 -464.249,E2 -464.249} C_VEL
LIN {X 0,Y 608.484,Z 483.747,A -85,B 0,C 180,E1 -467.128,E2 -467.128} C_VEL
LIN {X 0,Y 608.489,Z 468.447,A -85,B 0,C 180,E1 -469.92,E2 -469.92} C_VEL
LIN {X 0,Y 608.525,Z 454.586,A -85,B 0,C 180,E1 -472.491,E2 -472.491} C_VEL
LIN {X 0,Y 608.563,Z 439.76,A -85,B 0,C 180,E1 -475.295,E2 -475.295} C_VEL
LIN {X 0,Y 608.573,Z 426.373,A -85,B 0,C 180,E1 -477.884,E2 -477.884} C_VEL
LIN {X 0,Y 608.609,Z 412.986,A -85,B 0,C 180,E1 -480.536,E2 -480.536} C_VEL
LIN {X 0,Y 608.656,Z 399.592,A -85,B 0,C 180,E1 -483.261,E2 -483.261} C_VEL
LIN {X 0,Y 608.626,Z 384.352,A -85,B 0,C 180,E1 -486.283,E2 -486.283} C_VEL
LIN {X 0,Y 608.548,Z 373.744,A -85,B 0,C 180,E1 -488.479,E2 -488.479} C_VEL
LIN {X 0,Y 608.475,Z 373.313,A -85,B 0,C 180,E1 -488.586,E2 -488.586} C_VEL
LIN {X 0,Y 608.456,Z 373.315,A -85,B 0,C 180,E1 -491.342,E2 -491.342} C_VEL
LIN {X 0,Y 608.448,Z 373.316,A -85,B 0,C 180,E1 -494.263,E2 -494.263} C_VEL
LIN {X 0,Y 608.453,Z 373.313,A -85,B 0,C 180,E1 -497.04,E2 -497.04} C_VEL
LIN {X 0,Y 608.451,Z 373.322,A -85,B 0,C 180,E1 -499.697,E2 -499.697} C_VEL
LIN {X 0,Y 608.468,Z 373.313,A -85,B 0,C 180,E1 -502.254,E2 -502.254} C_VEL
LIN {X 0,Y 608.469,Z 373.312,A -85,B 0,C 180,E1 -505.09,E2 -505.09} C_VEL
LIN {X 0,Y 608.468,Z 373.317,A -85,B 0,C 180,E1 -507.906,E2 -507.906} C_VEL
LIN {X 0,Y 608.462,Z 373.313,A -85,B 0,C 180,E1 -510.22,E2 -510.22} C_VEL
LIN {X 0,Y 608.475,Z 373.31,A -85,B 0,C 180,E1 -512.791,E2 -512.791} C_VEL
LIN {X 0,Y 608.449,Z 373.32,A -85,B 0,C 180,E1 -515.429,E2 -515.429} C_VEL
LIN {X 0,Y 608.471,Z 373.311,A -85,B 0,C 180,E1 -518.309,E2 -518.309} C_VEL
LIN {X 0,Y 608.465,Z 373.316,A -85,B 0,C 180,E1 -521.282,E2 -521.282} C_VEL
LIN {X 0,Y 608.456,Z 373.317,A -85,B 0,C 180,E1 -523.906,E2 -523.906} C_VEL
LIN {X 0,Y 608.46,Z 373.311,A -85,B 0,C 180,E1 -526.644,E2 -526.644} C_VEL
LIN {X 0,Y 608.466,Z 373.318,A -85,B 0,C 180,E1 -529.35,E2 -529.35} C_VEL
LIN {X 0,Y 608.47,Z 373.313,A -85,B 0,C 180,E1 -532.033,E2 -532.033} C_VEL
LIN {X 0,Y 608.462,Z 373.311,A -85,B 0,C 180,E1 -534.698,E2 -534.698} C_VEL
LIN {X 0,Y 608.481,Z 373.317,A -85,B 0,C 180,E1 -537.352,E2 -537.352} C_VEL
LIN {X 0,Y 608.468,Z 373.313,A -85,B 0,C 180,E1 -540,E2 -540} C_VEL
LIN {X 0,Y 608.479,Z 373.309,A -85,B 0,C 180,E1 -542.648,E2 -542.648} C_VEL
LIN {X 0,Y 608.464,Z 373.319,A -85,B 0,C 180,E1 -545.302,E2 -545.302} C_VEL
LIN {X 0,Y 608.47,Z 373.312,A -85,B 0,C 180,E1 -547.967,E2 -547.967} C_VEL
LIN {X 0,Y 608.455,Z 373.318,A -85,B 0,C 180,E1 -549.472,E2 -549.472} C_VEL
LIN {X 0,Y 607.773,Z 373.399,A -85,B 0,C 180,E1 -550.024,E2 -550.024} C_VEL
LIN {X 0,Y 604.915,Z 373.756,A -85,B 0,C 180,E1 -550.921,E2 -550.921} C_VEL
LIN {X 0,Y 602.512,Z 374.059,A -85,B 0,C 180,E1 -551.643,E2 -551.643} C_VEL
LIN {X 0,Y 601.486,Z 374.181,A -85,B 0,C 180,E1 -552.2,E2 -552.2} C_VEL
LIN {X 0,Y 601.404,Z 374.19,A -85,B 0,C 180,E1 -552.388,E2 -552.388} C_VEL
LIN {X 0,Y 601.428,Z 374.191,A -85,B 0,C 180,E1 -554.897,E2 -554.897} C_VEL
LIN {X 0,Y 601.429,Z 374.192,A -85,B 0,C 180,E1 -556.986,E2 -556.986} C_VEL
LIN {X 0,Y 601.403,Z 374.194,A -85,B 0,C 180,E1 -559.81,E2 -559.81} C_VEL
LIN {X 0,Y 601.405,Z 374.192,A -85,B 0,C 180,E1 -562.684,E2 -562.684} C_VEL
LIN {X 0,Y 601.399,Z 374.195,A -85,B 0,C 180,E1 -564.879,E2 -564.879} C_VEL
LIN {X 0,Y 601.418,Z 374.19,A -85,B 0,C 180,E1 -567.868,E2 -567.868} C_VEL
LIN {X 0,Y 601.42,Z 374.189,A -85,B 0,C 180,E1 -570.165,E2 -570.165} C_VEL
LIN {X 0,Y 601.424,Z 374.191,A -85,B 0,C 180,E1 -572.718,E2 -572.718} C_VEL
LIN {X 0,Y 601.406,Z 374.199,A -85,B 0,C 180,E1 -575.115,E2 -575.115} C_VEL
LIN {X 0,Y 601.431,Z 374.194,A -85,B 0,C 180,E1 -577.42,E2 -577.42} C_VEL
LIN {X 0,Y 601.408,Z 374.19,A -85,B 0,C 180,E1 -579.996,E2 -579.996} C_VEL
LIN {X 0,Y 601.433,Z 374.19,A -85,B 0,C 180,E1 -582.669,E2 -582.669} C_VEL
LIN {X 0,Y 601.421,Z 374.193,A -85,B 0,C 180,E1 -585.483,E2 -585.483} C_VEL
LIN {X 0,Y 601.422,Z 374.189,A -85,B 0,C 180,E1 -588.408,E2 -588.408} C_VEL
LIN {X 0,Y 601.437,Z 374.193,A -85,B 0,C 180,E1 -590.877,E2 -590.877} C_VEL
LIN {X 0,Y 601.442,Z 374.187,A -85,B 0,C 180,E1 -593.735,E2 -593.735} C_VEL
LIN {X 0,Y 601.431,Z 374.187,A -85,B 0,C 180,E1 -596.065,E2 -596.065} C_VEL
LIN {X 0,Y 601.43,Z 374.198,A -85,B 0,C 180,E1 -599.06,E2 -599.06} C_VEL
LIN {X 0,Y 601.429,Z 374.192,A -85,B 0,C 180,E1 -601.374,E2 -601.374} C_VEL
LIN {X 0,Y 601.402,Z 374.192,A -85,B 0,C 180,E1 -603.637,E2 -603.637} C_VEL
LIN {X 0,Y 601.42,Z 374.193,A -85,B 0,C 180,E1 -606.591,E2 -606.591} C_VEL
LIN {X 0,Y 601.429,Z 374.19,A -85,B 0,C 180,E1 -609.479,E2 -609.479} C_VEL
LIN {X 0,Y 601.4,Z 374.192,A -85,B 0,C 180,E1 -612.313,E2 -612.313} C_VEL
LIN {X 0,Y 601.416,Z 374.191,A -85,B 0,C 180,E1 -614.41,E2 -614.41} C_VEL
LIN {X 0,Y 601.319,Z 374.553,A -85,B 0,C 180,E1 -615.793,E2 -615.793} C_VEL
LIN {X 0,Y 601.319,Z 378.022,A -85,B 0,C 180,E1 -618.541,E2 -618.541} C_VEL
LIN {X 0,Y 601.336,Z 381.497,A -85,B 0,C 180,E1 -621.198,E2 -621.198} C_VEL
LIN {X 0,Y 601.595,Z 391.212,A -85,B 0,C 180,E1 -621.414,E2 -621.414} C_VEL
LIN {X 0,Y 601.559,Z 403.946,A -85,B 0,C 180,E1 -621.815,E2 -621.815} C_VEL
LIN {X 0,Y 601.508,Z 416.585,A -85,B 0,C 180,E1 -622.363,E2 -622.363} C_VEL
LIN {X 0,Y 601.477,Z 427.126,A -85,B 0,C 180,E1 -622.954,E2 -622.954} C_VEL
LIN {X 0,Y 601.479,Z 437.416,A -85,B 0,C 180,E1 -623.67,E2 -623.67} C_VEL
LIN {X 0,Y 601.431,Z 446.755,A -85,B 0,C 180,E1 -624.469,E2 -624.469} C_VEL
LIN {X 0,Y 601.379,Z 456.337,A -85,B 0,C 180,E1 -625.476,E2 -625.476} C_VEL
LIN {X 0,Y 601.361,Z 463.994,A -85,B 0,C 180,E1 -626.483,E2 -626.483} C_VEL
LIN {X 0,Y 601.367,Z 471.053,A -85,B 0,C 180,E1 -627.657,E2 -627.657} C_VEL
LIN {X 0,Y 601.352,Z 475.758,A -85,B 0,C 180,E1 -628.661,E2 -628.661} C_VEL
LIN {X 0,Y 601.368,Z 479.364,A -85,B 0,C 180,E1 -629.666,E2 -629.666} C_VEL
LIN {X 0,Y 601.338,Z 481.975,A -85,B 0,C 180,E1 -630.67,E2 -630.67} C_VEL
LIN {X 0,Y 601.35,Z 483.201,A -85,B 0,C 180,E1 -631.34,E2 -631.34} C_VEL
LIN {X 0,Y 601.343,Z 484.027,A -85,B 0,C 180,E1 -632.01,E2 -632.01} C_VEL
LIN {X 0,Y 601.338,Z 484.435,A -85,B 0,C 180,E1 -633.351,E2 -633.351} C_VEL
LIN {X 0,Y 601.342,Z 484.07,A -85,B 0,C 180,E1 -634.022,E2 -634.022} C_VEL
LIN {X 0,Y 601.328,Z 483.294,A -85,B 0,C 180,E1 -634.693,E2 -634.693} C_VEL
LIN {X 0,Y 601.349,Z 482.091,A -85,B 0,C 180,E1 -635.365,E2 -635.365} C_VEL
LIN {X 0,Y 601.349,Z 478.862,A -85,B 0,C 180,E1 -636.583,E2 -636.583} C_VEL
LIN {X 0,Y 601.354,Z 474.506,A -85,B 0,C 180,E1 -637.725,E2 -637.725} C_VEL
LIN {X 0,Y 601.361,Z 468.412,A -85,B 0,C 180,E1 -638.909,E2 -638.909} C_VEL
LIN {X 0,Y 601.389,Z 461.725,A -85,B 0,C 180,E1 -639.926,E2 -639.926} C_VEL
LIN {X 0,Y 601.392,Z 452.989,A -85,B 0,C 180,E1 -640.993,E2 -640.993} C_VEL
LIN {X 0,Y 601.45,Z 444.832,A -85,B 0,C 180,E1 -641.8,E2 -641.8} C_VEL
LIN {X 0,Y 601.451,Z 434.232,A -85,B 0,C 180,E1 -642.656,E2 -642.656} C_VEL
LIN {X 0,Y 601.483,Z 423.702,A -85,B 0,C 180,E1 -643.343,E2 -643.343} C_VEL
LIN {X 0,Y 601.547,Z 412.518,A -85,B 0,C 180,E1 -643.922,E2 -643.922} C_VEL
LIN {X 0,Y 601.566,Z 399.884,A -85,B 0,C 180,E1 -644.418,E2 -644.418} C_VEL
LIN {X 0,Y 601.602,Z 386.637,A -85,B 0,C 180,E1 -644.785,E2 -644.785} C_VEL
LIN {X 0,Y 601.351,Z 381.408,A -85,B 0,C 180,E1 -644.899,E2 -644.899} C_VEL
LIN {X 0,Y 601.305,Z 377.842,A -85,B 0,C 180,E1 -647.692,E2 -647.692} C_VEL
LIN {X 0,Y 601.343,Z 374.266,A -85,B 0,C 180,E1 -650.525,E2 -650.525} C_VEL
LIN {X 0,Y 601.419,Z 374.193,A -85,B 0,C 180,E1 -652.683,E2 -652.683} C_VEL
LIN {X 0,Y 601.406,Z 374.198,A -85,B 0,C 180,E1 -654.879,E2 -654.879} C_VEL
LIN {X 0,Y 601.418,Z 374.193,A -85,B 0,C 180,E1 -657.362,E2 -657.362} C_VEL
LIN {X 0,Y 601.434,Z 374.188,A -85,B 0,C 180,E1 -660.164,E2 -660.164} C_VEL
LIN {X 0,Y 601.419,Z 374.198,A -85,B 0,C 180,E1 -662.714,E2 -662.714} C_VEL
LIN {X 0,Y 601.405,Z 374.195,A -85,B 0,C 180,E1 -665.113,E2 -665.113} C_VEL
LIN {X 0,Y 601.438,Z 374.187,A -85,B 0,C 180,E1 -667.419,E2 -667.419} C_VEL
LIN {X 0,Y 601.408,Z 374.192,A -85,B 0,C 180,E1 -669.996,E2 -669.996} C_VEL
LIN {X 0,Y 601.414,Z 374.196,A -85,B 0,C 180,E1 -672.67,E2 -672.67} C_VEL
LIN {X 0,Y 601.432,Z 374.187,A -85,B 0,C 180,E1 -675.482,E2 -675.482} C_VEL
LIN {X 0,Y 601.43,Z 374.195,A -85,B 0,C 180,E1 -678.407,E2 -678.407} C_VEL
LIN {X 0,Y 601.437,Z 374.186,A -85,B 0,C 180,E1 -680.875,E2 -680.875} C_VEL
LIN {X 0,Y 601.447,Z 374.19,A -85,B 0,C 180,E1 -683.734,E2 -683.734} C_VEL
LIN {X 0,Y 601.423,Z 374.189,A -85,B 0,C 180,E1 -686.686,E2 -686.686} C_VEL
LIN {X 0,Y 601.417,Z 374.189,A -85,B 0,C 180,E1 -689.058,E2 -689.058} C_VEL
LIN {X 0,Y 601.433,Z 374.189,A -85,B 0,C 180,E1 -691.373,E2 -691.373} C_VEL
LIN {X 0,Y 601.403,Z 374.199,A -85,B 0,C 180,E1 -693.636,E2 -693.636} C_VEL
LIN {X 0,Y 601.453,Z 374.192,A -85,B 0,C 180,E1 -695.859,E2 -695.859} C_VEL
LIN {X 0,Y 601.409,Z 374.19,A -85,B 0,C 180,E1 -698.761,E2 -698.761} C_VEL
LIN {X 0,Y 601.419,Z 374.198,A -85,B 0,C 180,E1 -701.608,E2 -701.608} C_VEL
LIN {X 0,Y 601.439,Z 374.192,A -85,B 0,C 180,E1 -703.713,E2 -703.713} C_VEL
LIN {X 0,Y 601.412,Z 374.191,A -85,B 0,C 180,E1 -706.484,E2 -706.484} C_VEL
LIN {X 0,Y 601.441,Z 374.319,A -85,B 0,C 180,E1 -707.097,E2 -707.097} C_VEL
LIN {X 0,Y 601.691,Z 379.841,A -85,B 0,C 180,E1 -707.263,E2 -707.263} C_VEL
LIN {X 0,Y 601.611,Z 393.802,A -85,B 0,C 180,E1 -707.776,E2 -707.776} C_VEL
LIN {X 0,Y 601.599,Z 406.304,A -85,B 0,C 180,E1 -708.374,E2 -708.374} C_VEL
LIN {X 0,Y 601.548,Z 418.053,A -85,B 0,C 180,E1 -709.071,E2 -709.071} C_VEL
LIN {X 0,Y 601.491,Z 429.591,A -85,B 0,C 180,E1 -709.906,E2 -709.906} C_VEL
LIN {X 0,Y 601.444,Z 441.117,A -85,B 0,C 180,E1 -710.923,E2 -710.923} C_VEL
LIN {X 0,Y 601.405,Z 450.567,A -85,B 0,C 180,E1 -711.939,E2 -711.939} C_VEL
LIN {X 0,Y 601.387,Z 459.586,A -85,B 0,C 180,E1 -713.12,E2 -713.12} C_VEL
LIN {X 0,Y 601.373,Z 466.867,A -85,B 0,C 180,E1 -714.299,E2 -714.299} C_VEL
LIN {X 0,Y 601.356,Z 473.409,A -85,B 0,C 180,E1 -715.643,E2 -715.643} C_VEL
LIN {X 0,Y 601.346,Z 478.316,A -85,B 0,C 180,E1 -716.985,E2 -716.985} C_VEL
LIN {X 0,Y 601.339,Z 481.032,A -85,B 0,C 180,E1 -717.991,E2 -717.991} C_VEL
LIN {X 0,Y 601.334,Z 483.397,A -85,B 0,C 180,E1 -719.33,E2 -719.33} C_VEL
LIN {X 0,Y 601.334,Z 484.421,A -85,B 0,C 180,E1 -720.669,E2 -720.669} C_VEL
LIN {X 0,Y 601.339,Z 484.125,A -85,B 0,C 180,E1 -722.009,E2 -722.009} C_VEL
LIN {X 0,Y 601.34,Z 482.511,A -85,B 0,C 180,E1 -723.35,E2 -723.35} C_VEL
LIN {X 0,Y 601.329,Z 479.531,A -85,B 0,C 180,E1 -724.693,E2 -724.693} C_VEL
LIN {X 0,Y 601.353,Z 475.098,A -85,B 0,C 180,E1 -726.038,E2 -726.038} C_VEL
LIN {X 0,Y 601.369,Z 470.691,A -85,B 0,C 180,E1 -727.048,E2 -727.048} C_VEL
LIN {X 0,Y 601.4,Z 464.307,A -85,B 0,C 180,E1 -728.23,E2 -728.23} C_VEL
LIN {X 0,Y 601.388,Z 456.377,A -85,B 0,C 180,E1 -729.416,E2 -729.416} C_VEL
LIN {X 0,Y 601.419,Z 448.078,A -85,B 0,C 180,E1 -730.435,E2 -730.435} C_VEL
LIN {X 0,Y 601.461,Z 438.075,A -85,B 0,C 180,E1 -731.457,E2 -731.457} C_VEL
LIN {X 0,Y 601.523,Z 426.886,A -85,B 0,C 180,E1 -732.397,E2 -732.397} C_VEL
LIN {X 0,Y 601.552,Z 414.358,A -85,B 0,C 180,E1 -733.255,E2 -733.255} C_VEL
LIN {X 0,Y 601.602,Z 402.365,A -85,B 0,C 180,E1 -733.919,E2 -733.919} C_VEL
LIN {X 0,Y 601.655,Z 389.077,A -85,B 0,C 180,E1 -734.502,E2 -734.502} C_VEL
LIN {X 0,Y 601.59,Z 375.06,A -85,B 0,C 180,E1 -734.968,E2 -734.968} C_VEL
LIN {X 0,Y 601.425,Z 374.196,A -85,B 0,C 180,E1 -735.005,E2 -735.005} C_VEL
LIN {X 0,Y 601.404,Z 374.2,A -85,B 0,C 180,E1 -737.688,E2 -737.688} C_VEL
LIN {X 0,Y 601.43,Z 374.196,A -85,B 0,C 180,E1 -740.522,E2 -740.522} C_VEL
LIN {X 0,Y 601.427,Z 374.194,A -85,B 0,C 180,E1 -743.41,E2 -743.41} C_VEL
LIN {X 0,Y 601.404,Z 374.199,A -85,B 0,C 180,E1 -746.364,E2 -746.364} C_VEL
LIN {X 0,Y 601.439,Z 374.194,A -85,B 0,C 180,E1 -748.789,E2 -748.789} C_VEL
LIN {X 0,Y 601.423,Z 374.198,A -85,B 0,C 180,E1 -751.455,E2 -751.455} C_VEL
LIN {X 0,Y 601.431,Z 374.197,A -85,B 0,C 180,E1 -754.118,E2 -754.118} C_VEL
LIN {X 0,Y 601.439,Z 374.193,A -85,B 0,C 180,E1 -757.382,E2 -757.382} C_VEL
LIN {X 0,Y 601.404,Z 374.198,A -85,B 0,C 180,E1 -759.996,E2 -759.996} C_VEL
LIN {X 0,Y 601.418,Z 374.198,A -85,B 0,C 180,E1 -762.67,E2 -762.67} C_VEL
LIN {X 0,Y 601.401,Z 374.2,A -85,B 0,C 180,E1 -765.479,E2 -765.479} C_VEL
LIN {X 0,Y 601.427,Z 374.195,A -85,B 0,C 180,E1 -768.407,E2 -768.407} C_VEL
LIN {X 0,Y 601.437,Z 374.194,A -85,B 0,C 180,E1 -770.875,E2 -770.875} C_VEL
LIN {X 0,Y 601.431,Z 374.24,A -85,B 0,C 180,E1 -772.052,E2 -772.052} C_VEL
LIN {X 0,Y 601.511,Z 386.552,A -85,B 0,C 180,E1 -774.253,E2 -774.253} C_VEL
LIN {X 0,Y 601.772,Z 405.244,A -85,B 0,C 180,E1 -777.505,E2 -777.505} C_VEL
LIN {X 0,Y 601.717,Z 418.715,A -85,B 0,C 180,E1 -780.238,E2 -780.238} C_VEL
LIN {X 0,Y 601.64,Z 432.102,A -85,B 0,C 180,E1 -782.898,E2 -782.898} C_VEL
LIN {X 0,Y 601.589,Z 446.416,A -85,B 0,C 180,E1 -785.675,E2 -785.675} C_VEL
LIN {X 0,Y 601.531,Z 460.789,A -85,B 0,C 180,E1 -788.405,E2 -788.405} C_VEL
LIN {X 0,Y 601.489,Z 476.789,A -85,B 0,C 180,E1 -791.386,E2 -791.386} C_VEL
LIN {X 0,Y 601.431,Z 491.389,A -85,B 0,C 180,E1 -794.061,E2 -794.061} C_VEL
LIN {X 0,Y 601.443,Z 499.979,A -85,B 0,C 180,E1 -795.591,E2 -795.591} C_VEL
LIN {X 0,Y 601.748,Z 506.768,A -85,B 0,C 180,E1 -795.689,E2 -795.689} C_VEL
LIN {X 0,Y 601.703,Z 521.088,A -85,B 0,C 180,E1 -795.973,E2 -795.973} C_VEL
LIN {X 0,Y 601.653,Z 534.931,A -85,B 0,C 180,E1 -796.387,E2 -796.387} C_VEL
LIN {X 0,Y 601.631,Z 548.079,A -85,B 0,C 180,E1 -796.918,E2 -796.918} C_VEL
LIN {X 0,Y 601.568,Z 561.256,A -85,B 0,C 180,E1 -797.603,E2 -797.603} C_VEL
LIN {X 0,Y 601.511,Z 573.141,A -85,B 0,C 180,E1 -798.372,E2 -798.372} C_VEL
LIN {X 0,Y 601.489,Z 583.985,A -85,B 0,C 180,E1 -799.225,E2 -799.225} C_VEL
LIN {X 0,Y 601.422,Z 594.702,A -85,B 0,C 180,E1 -800.244,E2 -800.244} C_VEL
LIN {X 0,Y 601.407,Z 603.552,A -85,B 0,C 180,E1 -801.261,E2 -801.261} C_VEL
LIN {X 0,Y 601.406,Z 612.035,A -85,B 0,C 180,E1 -802.445,E2 -802.445} C_VEL
LIN {X 0,Y 601.361,Z 618.751,A -85,B 0,C 180,E1 -803.604,E2 -803.604} C_VEL
LIN {X 0,Y 601.355,Z 623.565,A -85,B 0,C 180,E1 -804.635,E2 -804.635} C_VEL
LIN {X 0,Y 601.343,Z 628.44,A -85,B 0,C 180,E1 -805.978,E2 -805.978} C_VEL
LIN {X 0,Y 601.324,Z 631.83,A -85,B 0,C 180,E1 -807.32,E2 -807.32} C_VEL
LIN {X 0,Y 601.342,Z 633.83,A -85,B 0,C 180,E1 -808.66,E2 -808.66} C_VEL
LIN {X 0,Y 601.333,Z 634.5,A -85,B 0,C 180,E1 -809.999,E2 -809.999} C_VEL
LIN {X 0,Y 601.342,Z 633.832,A -85,B 0,C 180,E1 -811.339,E2 -811.339} C_VEL
LIN {X 0,Y 601.323,Z 631.833,A -85,B 0,C 180,E1 -812.679,E2 -812.679} C_VEL
LIN {X 0,Y 601.343,Z 628.444,A -85,B 0,C 180,E1 -814.02,E2 -814.02} C_VEL
LIN {X 0,Y 601.355,Z 623.571,A -85,B 0,C 180,E1 -815.364,E2 -815.364} C_VEL
LIN {X 0,Y 601.372,Z 617.625,A -85,B 0,C 180,E1 -816.605,E2 -816.605} C_VEL
LIN {X 0,Y 601.385,Z 610.924,A -85,B 0,C 180,E1 -817.723,E2 -817.723} C_VEL
LIN {X 0,Y 601.411,Z 602.205,A -85,B 0,C 180,E1 -818.907,E2 -818.907} C_VEL
LIN {X 0,Y 601.432,Z 593.09,A -85,B 0,C 180,E1 -819.924,E2 -819.924} C_VEL
LIN {X 0,Y 601.496,Z 582.832,A -85,B 0,C 180,E1 -820.876,E2 -820.876} C_VEL
LIN {X 0,Y 601.534,Z 571.983,A -85,B 0,C 180,E1 -821.712,E2 -821.712} C_VEL
LIN {X 0,Y 601.564,Z 559.791,A -85,B 0,C 180,E1 -822.481,E2 -822.481} C_VEL
LIN {X 0,Y 601.636,Z 546.147,A -85,B 0,C 180,E1 -823.166,E2 -823.166} C_VEL
LIN {X 0,Y 601.673,Z 531.887,A -85,B 0,C 180,E1 -823.714,E2 -823.714} C_VEL
LIN {X 0,Y 601.692,Z 518.057,A -85,B 0,C 180,E1 -824.098,E2 -824.098} C_VEL
LIN {X 0,Y 601.762,Z 503.894,A -85,B 0,C 180,E1 -824.351,E2 -824.351} C_VEL
LIN {X 0,Y 601.422,Z 499.706,A -85,B 0,C 180,E1 -824.431,E2 -824.431} C_VEL
LIN {X 0,Y 601.474,Z 483.747,A -85,B 0,C 180,E1 -827.334,E2 -827.334} C_VEL
LIN {X 0,Y 601.5,Z 470.36,A -85,B 0,C 180,E1 -829.805,E2 -829.805} C_VEL
LIN {X 0,Y 601.548,Z 455.06,A -85,B 0,C 180,E1 -832.677,E2 -832.677} C_VEL
LIN {X 0,Y 601.624,Z 439.76,A -85,B 0,C 180,E1 -835.608,E2 -835.608} C_VEL
LIN {X 0,Y 601.658,Z 426.373,A -85,B 0,C 180,E1 -838.233,E2 -838.233} C_VEL
LIN {X 0,Y 601.75,Z 412.986,A -85,B 0,C 180,E1 -840.922,E2 -840.922} C_VEL
LIN {X 0,Y 601.725,Z 402.737,A -85,B 0,C 180,E1 -842.982,E2 -842.982} C_VEL
LIN {X 0,Y 601.721,Z 387.573,A -85,B 0,C 180,E1 -846.018,E2 -846.018} C_VEL
LIN {X 0,Y 601.795,Z 376.888,A -85,B 0,C 180,E1 -848.238,E2 -848.238} C_VEL
LIN {X 0,Y 601.424,Z 374.194,A -85,B 0,C 180,E1 -848.863,E2 -848.863} C_VEL
LIN {X 0,Y 601.42,Z 374.199,A -85,B 0,C 180,E1 -851.764,E2 -851.764} C_VEL
LIN {X 0,Y 601.417,Z 374.19,A -85,B 0,C 180,E1 -854.534,E2 -854.534} C_VEL
LIN {X 0,Y 601.433,Z 374.191,A -85,B 0,C 180,E1 -857.405,E2 -857.405} C_VEL
LIN {X 0,Y 601.433,Z 374.188,A -85,B 0,C 180,E1 -860.463,E2 -860.463} C_VEL
LIN {X 0,Y 601.406,Z 374.195,A -85,B 0,C 180,E1 -863.417,E2 -863.417} C_VEL
LIN {X 0,Y 601.427,Z 374.192,A -85,B 0,C 180,E1 -866.063,E2 -866.063} C_VEL
LIN {X 0,Y 601.434,Z 374.187,A -85,B 0,C 180,E1 -868.541,E2 -868.541} C_VEL
LIN {X 0,Y 601.43,Z 374.193,A -85,B 0,C 180,E1 -871.373,E2 -871.373} C_VEL
LIN {X 0,Y 601.401,Z 374.202,A -85,B 0,C 180,E1 -873.636,E2 -873.636} C_VEL
LIN {X 0,Y 601.413,Z 374.189,A -85,B 0,C 180,E1 -876.589,E2 -876.589} C_VEL
LIN {X 0,Y 601.427,Z 374.196,A -85,B 0,C 180,E1 -879.478,E2 -879.478} C_VEL
LIN {X 0,Y 601.395,Z 374.193,A -85,B 0,C 180,E1 -882.312,E2 -882.312} C_VEL
LIN {X 0,Y 601.411,Z 374.19,A -85,B 0,C 180,E1 -884.409,E2 -884.409} C_VEL
LIN {X 0,Y 601.418,Z 374.193,A -85,B 0,C 180,E1 -887.172,E2 -887.172} C_VEL
LIN {X 0,Y 601.429,Z 374.192,A -85,B 0,C 180,E1 -889.905,E2 -889.905} C_VEL
LIN {X 0,Y 601.445,Z 374.185,A -85,B 0,C 180,E1 -892.615,E2 -892.615} C_VEL
LIN {X 0,Y 601.427,Z 374.195,A -85,B 0,C 180,E1 -895.308,E2 -895.308} C_VEL
LIN {X 0,Y 601.418,Z 374.191,A -85,B 0,C 180,E1 -897.991,E2 -897.991} C_VEL
LIN {X 0,Y 601.449,Z 374.185,A -85,B 0,C 180,E1 -900.67,E2 -900.67} C_VEL
LIN {X 0,Y 601.429,Z 374.197,A -85,B 0,C 180,E1 -903.35,E2 -903.35} C_VEL
LIN {X 0,Y 601.404,Z 374.192,A -85,B 0,C 180,E1 -906.037,E2 -906.037} C_VEL
LIN {X 0,Y 601.434,Z 374.188,A -85,B 0,C 180,E1 -908.738,E2 -908.738} C_VEL
LIN {X 0,Y 601.428,Z 374.197,A -85,B 0,C 180,E1 -911.458,E2 -911.458} C_VEL
LIN {X 0,Y 601.404,Z 374.19,A -85,B 0,C 180,E1 -912.388,E2 -912.388} C_VEL
LIN {X 0,Y 600.744,Z 374.278,A -85,B 0,C 180,E1 -912.947,E2 -912.947} C_VEL
LIN {X 0,Y 597.894,Z 374.632,A -85,B 0,C 180,E1 -913.855,E2 -913.855} C_VEL
LIN {X 0,Y 595.482,Z 374.934,A -85,B 0,C 180,E1 -914.585,E2 -914.585} C_VEL
LIN {X 0,Y 594.444,Z 375.065,A -85,B 0,C 180,E1 -915.149,E2 -915.149} C_VEL
LIN {X 0,Y 594.358,Z 375.072,A -85,B 0,C 180,E1 -915.34,E2 -915.34} C_VEL
LIN {X 0,Y 594.376,Z 375.068,A -85,B 0,C 180,E1 -917.905,E2 -917.905} C_VEL
LIN {X 0,Y 594.377,Z 375.07,A -85,B 0,C 180,E1 -920.919,E2 -920.919} C_VEL
LIN {X 0,Y 594.384,Z 375.069,A -85,B 0,C 180,E1 -923.705,E2 -923.705} C_VEL
LIN {X 0,Y 594.384,Z 375.067,A -85,B 0,C 180,E1 -926.7,E2 -926.7} C_VEL
LIN {X 0,Y 594.377,Z 375.072,A -85,B 0,C 180,E1 -928.999,E2 -928.999} C_VEL
LIN {X 0,Y 594.387,Z 375.069,A -85,B 0,C 180,E1 -931.647,E2 -931.647} C_VEL
LIN {X 0,Y 594.388,Z 375.066,A -85,B 0,C 180,E1 -934.58,E2 -934.58} C_VEL
LIN {X 0,Y 594.382,Z 375.074,A -85,B 0,C 180,E1 -937.087,E2 -937.087} C_VEL
LIN {X 0,Y 594.371,Z 375.069,A -85,B 0,C 180,E1 -939.776,E2 -939.776} C_VEL
LIN {X 0,Y 594.384,Z 375.066,A -85,B 0,C 180,E1 -942.375,E2 -942.375} C_VEL
LIN {X 0,Y 594.359,Z 375.078,A -85,B 0,C 180,E1 -945.192,E2 -945.192} C_VEL
LIN {X 0,Y 594.364,Z 375.07,A -85,B 0,C 180,E1 -947.626,E2 -947.626} C_VEL
LIN {X 0,Y 594.391,Z 375.065,A -85,B 0,C 180,E1 -950.322,E2 -950.322} C_VEL
LIN {X 0,Y 594.385,Z 375.073,A -85,B 0,C 180,E1 -952.915,E2 -952.915} C_VEL
LIN {X 0,Y 594.383,Z 375.066,A -85,B 0,C 180,E1 -955.862,E2 -955.862} C_VEL
LIN {X 0,Y 594.39,Z 375.069,A -85,B 0,C 180,E1 -958.652,E2 -958.652} C_VEL
LIN {X 0,Y 594.383,Z 375.075,A -85,B 0,C 180,E1 -961.043,E2 -961.043} C_VEL
LIN {X 0,Y 594.387,Z 375.065,A -85,B 0,C 180,E1 -963.978,E2 -963.978} C_VEL
LIN {X 0,Y 594.389,Z 375.066,A -85,B 0,C 180,E1 -966.297,E2 -966.297} C_VEL
LIN {X 0,Y 594.403,Z 375.069,A -85,B 0,C 180,E1 -969.225,E2 -969.225} C_VEL
LIN {X 0,Y 594.357,Z 375.069,A -85,B 0,C 180,E1 -972.096,E2 -972.096} C_VEL
LIN {X 0,Y 594.368,Z 375.068,A -85,B 0,C 180,E1 -974.22,E2 -974.22} C_VEL
LIN {X 0,Y 594.262,Z 375.088,A -85,B 0,C 180,E1 -975.877,E2 -975.877} C_VEL
LIN {X 0,Y 594.233,Z 378.07,A -85,B 0,C 180,E1 -978.402,E2 -978.402} C_VEL
LIN {X 0,Y 594.25,Z 381.412,A -85,B 0,C 180,E1 -981.05,E2 -981.05} C_VEL
LIN {X 0,Y 594.623,Z 386.521,A -85,B 0,C 180,E1 -981.162,E2 -981.162} C_VEL
LIN {X 0,Y 594.609,Z 400.211,A -85,B 0,C 180,E1 -981.547,E2 -981.547} C_VEL
LIN {X 0,Y 594.565,Z 412.038,A -85,B 0,C 180,E1 -982.017,E2 -982.017} C_VEL
LIN {X 0,Y 594.482,Z 423.536,A -85,B 0,C 180,E1 -982.614,E2 -982.614} C_VEL
LIN {X 0,Y 594.453,Z 434.917,A -85,B 0,C 180,E1 -983.37,E2 -983.37} C_VEL
LIN {X 0,Y 594.385,Z 445.359,A -85,B 0,C 180,E1 -984.233,E2 -984.233} C_VEL
LIN {X 0,Y 594.347,Z 453.706,A -85,B 0,C 180,E1 -985.083,E2 -985.083} C_VEL
LIN {X 0,Y 594.315,Z 461.875,A -85,B 0,C 180,E1 -986.102,E2 -986.102} C_VEL
LIN {X 0,Y 594.319,Z 467.457,A -85,B 0,C 180,E1 -986.95,E2 -986.95} C_VEL
LIN {X 0,Y 594.257,Z 472.922,A -85,B 0,C 180,E1 -987.968,E2 -987.968} C_VEL
LIN {X 0,Y 594.25,Z 477.209,A -85,B 0,C 180,E1 -988.984,E2 -988.984} C_VEL
LIN {X 0,Y 594.238,Z 480.443,A -85,B 0,C 180,E1 -990.001,E2 -990.001} C_VEL
LIN {X 0,Y 594.25,Z 483.259,A -85,B 0,C 180,E1 -991.356,E2 -991.356} C_VEL
LIN {X 0,Y 594.241,Z 484.054,A -85,B 0,C 180,E1 -992.034,E2 -992.034} C_VEL
LIN {X 0,Y 594.258,Z 484.427,A -85,B 0,C 180,E1 -993.391,E2 -993.391} C_VEL
LIN {X 0,Y 594.255,Z 484.044,A -85,B 0,C 180,E1 -994.07,E2 -994.07} C_VEL
LIN {X 0,Y 594.227,Z 483.234,A -85,B 0,C 180,E1 -994.75,E2 -994.75} C_VEL
LIN {X 0,Y 594.263,Z 482.013,A -85,B 0,C 180,E1 -995.43,E2 -995.43} C_VEL
LIN {X 0,Y 594.264,Z 479.023,A -85,B 0,C 180,E1 -996.574,E2 -996.574} C_VEL
LIN {X 0,Y 594.281,Z 474.351,A -85,B 0,C 180,E1 -997.817,E2 -997.817} C_VEL
LIN {X 0,Y 594.293,Z 468.196,A -85,B 0,C 180,E1 -999.016,E2 -999.016} C_VEL
LIN {X 0,Y 594.327,Z 461.459,A -85,B 0,C 180,E1 -1000.046,E2 -1000.046} C_VEL
LIN {X 0,Y 594.336,Z 453.38,A -85,B 0,C 180,E1 -1001.045,E2 -1001.045} C_VEL
LIN {X 0,Y 594.395,Z 444.414,A -85,B 0,C 180,E1 -1001.942,E2 -1001.942} C_VEL
LIN {X 0,Y 594.449,Z 433.731,A -85,B 0,C 180,E1 -1002.808,E2 -1002.808} C_VEL
LIN {X 0,Y 594.474,Z 423.075,A -85,B 0,C 180,E1 -1003.503,E2 -1003.503} C_VEL
LIN {X 0,Y 594.543,Z 411.515,A -85,B 0,C 180,E1 -1004.097,E2 -1004.097} C_VEL
LIN {X 0,Y 594.625,Z 398.768,A -85,B 0,C 180,E1 -1004.59,E2 -1004.59} C_VEL
LIN {X 0,Y 594.665,Z 385.945,A -85,B 0,C 180,E1 -1004.94,E2 -1004.94} C_VEL
LIN {X 0,Y 594.242,Z 381.415,A -85,B 0,C 180,E1 -1005.038,E2 -1005.038} C_VEL
LIN {X 0,Y 594.204,Z 377.792,A -85,B 0,C 180,E1 -1007.91,E2 -1007.91} C_VEL
LIN {X 0,Y 594.219,Z 375.11,A -85,B 0,C 180,E1 -1010.06,E2 -1010.06} C_VEL
LIN {X 0,Y 594.362,Z 375.068,A -85,B 0,C 180,E1 -1012.234,E2 -1012.234} C_VEL
LIN {X 0,Y 594.395,Z 375.066,A -85,B 0,C 180,E1 -1014.446,E2 -1014.446} C_VEL
LIN {X 0,Y 594.387,Z 375.071,A -85,B 0,C 180,E1 -1016.7,E2 -1016.7} C_VEL
LIN {X 0,Y 594.386,Z 375.074,A -85,B 0,C 180,E1 -1018.999,E2 -1018.999} C_VEL
LIN {X 0,Y 594.381,Z 375.066,A -85,B 0,C 180,E1 -1021.642,E2 -1021.642} C_VEL
LIN {X 0,Y 594.387,Z 375.073,A -85,B 0,C 180,E1 -1024.58,E2 -1024.58} C_VEL
LIN {X 0,Y 594.393,Z 375.064,A -85,B 0,C 180,E1 -1027.608,E2 -1027.608} C_VEL
LIN {X 0,Y 594.373,Z 375.076,A -85,B 0,C 180,E1 -1030.567,E2 -1030.567} C_VEL
LIN {X 0,Y 594.371,Z 375.067,A -85,B 0,C 180,E1 -1033.3,E2 -1033.3} C_VEL
LIN {X 0,Y 594.388,Z 375.072,A -85,B 0,C 180,E1 -1036.159,E2 -1036.159} C_VEL
LIN {X 0,Y 594.38,Z 375.065,A -85,B 0,C 180,E1 -1039.178,E2 -1039.178} C_VEL
LIN {X 0,Y 594.392,Z 375.071,A -85,B 0,C 180,E1 -1042.059,E2 -1042.059} C_VEL
LIN {X 0,Y 594.357,Z 375.07,A -85,B 0,C 180,E1 -1044.676,E2 -1044.676} C_VEL
LIN {X 0,Y 594.382,Z 375.066,A -85,B 0,C 180,E1 -1047.088,E2 -1047.088} C_VEL
LIN {X 0,Y 594.389,Z 375.07,A -85,B 0,C 180,E1 -1049.672,E2 -1049.672} C_VEL
LIN {X 0,Y 594.379,Z 375.066,A -85,B 0,C 180,E1 -1052.539,E2 -1052.539} C_VEL
LIN {X 0,Y 594.374,Z 375.067,A -85,B 0,C 180,E1 -1054.807,E2 -1054.807} C_VEL
LIN {X 0,Y 594.365,Z 375.072,A -85,B 0,C 180,E1 -1057.265,E2 -1057.265} C_VEL
LIN {X 0,Y 594.375,Z 375.07,A -85,B 0,C 180,E1 -1059.946,E2 -1059.946} C_VEL
LIN {X 0,Y 594.391,Z 375.066,A -85,B 0,C 180,E1 -1062.806,E2 -1062.806} C_VEL
LIN {X 0,Y 594.391,Z 375.068,A -85,B 0,C 180,E1 -1065.826,E2 -1065.826} C_VEL
LIN {X 0,Y 594.393,Z 375.157,A -85,B 0,C 180,E1 -1066.952,E2 -1066.952} C_VEL
LIN {X 0,Y 594.79,Z 378.817,A -85,B 0,C 180,E1 -1067.07,E2 -1067.07} C_VEL
LIN {X 0,Y 594.732,Z 392.077,A -85,B 0,C 180,E1 -1067.545,E2 -1067.545} C_VEL
LIN {X 0,Y 594.636,Z 404.974,A -85,B 0,C 180,E1 -1068.149,E2 -1068.149} C_VEL
LIN {X 0,Y 594.55,Z 416.872,A -85,B 0,C 180,E1 -1068.849,E2 -1068.849} C_VEL
LIN {X 0,Y 594.481,Z 428.693,A -85,B 0,C 180,E1 -1069.699,E2 -1069.699} C_VEL
LIN {X 0,Y 594.439,Z 439.481,A -85,B 0,C 180,E1 -1070.644,E2 -1070.644} C_VEL
LIN {X 0,Y 594.371,Z 449.2,A -85,B 0,C 180,E1 -1071.671,E2 -1071.671} C_VEL
LIN {X 0,Y 594.346,Z 457.265,A -85,B 0,C 180,E1 -1072.697,E2 -1072.697} C_VEL
LIN {X 0,Y 594.288,Z 464.994,A -85,B 0,C 180,E1 -1073.89,E2 -1073.89} C_VEL
LIN {X 0,Y 594.256,Z 470.415,A -85,B 0,C 180,E1 -1074.911,E2 -1074.911} C_VEL
LIN {X 0,Y 594.288,Z 476.11,A -85,B 0,C 180,E1 -1076.271,E2 -1076.271} C_VEL
LIN {X 0,Y 594.232,Z 479.362,A -85,B 0,C 180,E1 -1077.288,E2 -1077.288} C_VEL
LIN {X 0,Y 594.242,Z 482.398,A -85,B 0,C 180,E1 -1078.644,E2 -1078.644} C_VEL
LIN {X 0,Y 594.234,Z 484.076,A -85,B 0,C 180,E1 -1080,E2 -1080} C_VEL
LIN {X 0,Y 594.247,Z 484.438,A -85,B 0,C 180,E1 -1081.355,E2 -1081.355} C_VEL
LIN {X 0,Y 594.222,Z 483.478,A -85,B 0,C 180,E1 -1082.711,E2 -1082.711} C_VEL
LIN {X 0,Y 594.253,Z 481.175,A -85,B 0,C 180,E1 -1084.069,E2 -1084.069} C_VEL
LIN {X 0,Y 594.27,Z 477.453,A -85,B 0,C 180,E1 -1085.429,E2 -1085.429} C_VEL
LIN {X 0,Y 594.277,Z 472.235,A -85,B 0,C 180,E1 -1086.792,E2 -1086.792} C_VEL
LIN {X 0,Y 594.304,Z 467.166,A -85,B 0,C 180,E1 -1087.816,E2 -1087.816} C_VEL
LIN {X 0,Y 594.34,Z 459.919,A -85,B 0,C 180,E1 -1089.014,E2 -1089.014} C_VEL
LIN {X 0,Y 594.347,Z 452.313,A -85,B 0,C 180,E1 -1090.044,E2 -1090.044} C_VEL
LIN {X 0,Y 594.402,Z 443.16,A -85,B 0,C 180,E1 -1091.079,E2 -1091.079} C_VEL
LIN {X 0,Y 594.46,Z 434.083,A -85,B 0,C 180,E1 -1091.94,E2 -1091.94} C_VEL
LIN {X 0,Y 594.548,Z 422.035,A -85,B 0,C 180,E1 -1092.892,E2 -1092.892} C_VEL
LIN {X 0,Y 594.598,Z 409.779,A -85,B 0,C 180,E1 -1093.674,E2 -1093.674} C_VEL
LIN {X 0,Y 594.681,Z 398.013,A -85,B 0,C 180,E1 -1094.284,E2 -1094.284} C_VEL
LIN {X 0,Y 594.767,Z 384.075,A -85,B 0,C 180,E1 -1094.849,E2 -1094.849} C_VEL
LIN {X 0,Y 594.636,Z 376.135,A -85,B 0,C 180,E1 -1095.104,E2 -1095.104} C_VEL
LIN {X 0,Y 594.421,Z 375.07,A -85,B 0,C 180,E1 -1095.164,E2 -1095.164} C_VEL
LIN {X 0,Y 594.384,Z 375.075,A -85,B 0,C 180,E1 -1097.904,E2 -1097.904} C_VEL
LIN {X 0,Y 594.38,Z 375.072,A -85,B 0,C 180,E1 -1100.916,E2 -1100.916} C_VEL
LIN {X 0,Y 594.397,Z 375.071,A -85,B 0,C 180,E1 -1103.704,E2 -1103.704} C_VEL
LIN {X 0,Y 594.387,Z 375.074,A -85,B 0,C 180,E1 -1106.699,E2 -1106.699} C_VEL
LIN {X 0,Y 594.383,Z 375.075,A -85,B 0,C 180,E1 -1108.998,E2 -1108.998} C_VEL
LIN {X 0,Y 594.381,Z 375.075,A -85,B 0,C 180,E1 -1111.643,E2 -1111.643} C_VEL
LIN {X 0,Y 594.379,Z 375.072,A -85,B 0,C 180,E1 -1114.58,E2 -1114.58} C_VEL
LIN {X 0,Y 594.394,Z 375.072,A -85,B 0,C 180,E1 -1117.609,E2 -1117.609} C_VEL
LIN {X 0,Y 594.37,Z 375.075,A -85,B 0,C 180,E1 -1120.567,E2 -1120.567} C_VEL
LIN {X 0,Y 594.384,Z 375.072,A -85,B 0,C 180,E1 -1123.298,E2 -1123.298} C_VEL
LIN {X 0,Y 594.363,Z 375.075,A -85,B 0,C 180,E1 -1126.161,E2 -1126.161} C_VEL
LIN {X 0,Y 594.383,Z 375.072,A -85,B 0,C 180,E1 -1128.536,E2 -1128.536} C_VEL
LIN {X 0,Y 594.389,Z 375.074,A -85,B 0,C 180,E1 -1131.295,E2 -1131.295} C_VEL
LIN {X 0,Y 594.411,Z 375.176,A -85,B 0,C 180,E1 -1131.953,E2 -1131.953} C_VEL
LIN {X 0,Y 594.465,Z 385.032,A -85,B 0,C 180,E1 -1133.763,E2 -1133.763} C_VEL
LIN {X 0,Y 594.711,Z 404.965,A -85,B 0,C 180,E1 -1137.272,E2 -1137.272} C_VEL
LIN {X 0,Y 594.868,Z 412.939,A -85,B 0,C 180,E1 -1138.679,E2 -1138.679} C_VEL
LIN {X 0,Y 594.784,Z 426.365,A -85,B 0,C 180,E1 -1141.409,E2 -1141.409} C_VEL
LIN {X 0,Y 594.689,Z 439.752,A -85,B 0,C 180,E1 -1144.07,E2 -1144.07} C_VEL
LIN {X 0,Y 594.593,Z 453.139,A -85,B 0,C 180,E1 -1146.673,E2 -1146.673} C_VEL
LIN {X 0,Y 594.516,Z 468.439,A -85,B 0,C 180,E1 -1149.59,E2 -1149.59} C_VEL
LIN {X 0,Y 594.467,Z 483.739,A -85,B 0,C 180,E1 -1152.454,E2 -1152.454} C_VEL
LIN {X 0,Y 594.391,Z 499.784,A -85,B 0,C 180,E1 -1155.409,E2 -1155.409} C_VEL
LIN {X 0,Y 594.862,Z 504.511,A -85,B 0,C 180,E1 -1155.487,E2 -1155.487} C_VEL
LIN {X 0,Y 594.831,Z 518.846,A -85,B 0,C 180,E1 -1155.754,E2 -1155.754} C_VEL
LIN {X 0,Y 594.774,Z 532.182,A -85,B 0,C 180,E1 -1156.134,E2 -1156.134} C_VEL
LIN {X 0,Y 594.693,Z 546.114,A -85,B 0,C 180,E1 -1156.676,E2 -1156.676} C_VEL
LIN {X 0,Y 594.605,Z 559.766,A -85,B 0,C 180,E1 -1157.369,E2 -1157.369} C_VEL
LIN {X 0,Y 594.548,Z 571.961,A -85,B 0,C 180,E1 -1158.147,E2 -1158.147} C_VEL
LIN {X 0,Y 594.462,Z 582.799,A -85,B 0,C 180,E1 -1158.991,E2 -1158.991} C_VEL
LIN {X 0,Y 594.4,Z 593.075,A -85,B 0,C 180,E1 -1159.956,E2 -1159.956} C_VEL
LIN {X 0,Y 594.369,Z 602.193,A -85,B 0,C 180,E1 -1160.986,E2 -1160.986} C_VEL
LIN {X 0,Y 594.316,Z 610.915,A -85,B 0,C 180,E1 -1162.183,E2 -1162.183} C_VEL
LIN {X 0,Y 594.277,Z 618.134,A -85,B 0,C 180,E1 -1163.412,E2 -1163.412} C_VEL
LIN {X 0,Y 594.275,Z 623.565,A -85,B 0,C 180,E1 -1164.57,E2 -1164.57} C_VEL
LIN {X 0,Y 594.259,Z 628.44,A -85,B 0,C 180,E1 -1165.93,E2 -1165.93} C_VEL
LIN {X 0,Y 594.224,Z 631.83,A -85,B 0,C 180,E1 -1167.288,E2 -1167.288} C_VEL
LIN {X 0,Y 594.242,Z 633.83,A -85,B 0,C 180,E1 -1168.644,E2 -1168.644} C_VEL
LIN {X 0,Y 594.234,Z 634.5,A -85,B 0,C 180,E1 -1169.999,E2 -1169.999} C_VEL
LIN {X 0,Y 594.242,Z 633.832,A -85,B 0,C 180,E1 -1171.355,E2 -1171.355} C_VEL
LIN {X 0,Y 594.224,Z 631.833,A -85,B 0,C 180,E1 -1172.711,E2 -1172.711} C_VEL
LIN {X 0,Y 594.259,Z 628.444,A -85,B 0,C 180,E1 -1174.068,E2 -1174.068} C_VEL
LIN {X 0,Y 594.275,Z 623.571,A -85,B 0,C 180,E1 -1175.428,E2 -1175.428} C_VEL
LIN {X 0,Y 594.299,Z 618.036,A -85,B 0,C 180,E1 -1176.607,E2 -1176.607} C_VEL
LIN {X 0,Y 594.315,Z 610.924,A -85,B 0,C 180,E1 -1177.815,E2 -1177.815} C_VEL
LIN {X 0,Y 594.368,Z 602.205,A -85,B 0,C 180,E1 -1179.013,E2 -1179.013} C_VEL
LIN {X 0,Y 594.399,Z 593.089,A -85,B 0,C 180,E1 -1180.043,E2 -1180.043} C_VEL
LIN {X 0,Y 594.477,Z 582.709,A -85,B 0,C 180,E1 -1181.017,E2 -1181.017} C_VEL
LIN {X 0,Y 594.574,Z 570.717,A -85,B 0,C 180,E1 -1181.937,E2 -1181.937} C_VEL
LIN {X 0,Y 594.604,Z 558.227,A -85,B 0,C 180,E1 -1182.716,E2 -1182.716} C_VEL
LIN {X 0,Y 594.693,Z 546.149,A -85,B 0,C 180,E1 -1183.323,E2 -1183.323} C_VEL
LIN {X 0,Y 594.774,Z 532.207,A -85,B 0,C 180,E1 -1183.866,E2 -1183.866} C_VEL
LIN {X 0,Y 594.815,Z 518.309,A -85,B 0,C 180,E1 -1184.259,E2 -1184.259} C_VEL
LIN {X 0,Y 594.88,Z 503.814,A -85,B 0,C 180,E1 -1184.522,E2 -1184.522} C_VEL
LIN {X 0,Y 594.39,Z 499.805,A -85,B 0,C 180,E1 -1184.587,E2 -1184.587} C_VEL
LIN {X 0,Y 594.466,Z 483.747,A -85,B 0,C 180,E1 -1187.545,E2 -1187.545} C_VEL
LIN {X 0,Y 594.485,Z 470.36,A -85,B 0,C 180,E1 -1190.049,E2 -1190.049} C_VEL
LIN {X 0,Y 594.612,Z 455.06,A -85,B 0,C 180,E1 -1192.956,E2 -1192.956} C_VEL
LIN {X 0,Y 594.689,Z 439.76,A -85,B 0,C 180,E1 -1195.928,E2 -1195.928} C_VEL
LIN {X 0,Y 594.782,Z 426.373,A -85,B 0,C 180,E1 -1198.59,E2 -1198.59} C_VEL
LIN {X 0,Y 594.862,Z 412.948,A -85,B 0,C 180,E1 -1201.32,E2 -1201.32} C_VEL
LIN {X 0,Y 594.793,Z 399.493,A -85,B 0,C 180,E1 -1203.961,E2 -1203.961} C_VEL
LIN {X 0,Y 594.889,Z 385.947,A -85,B 0,C 180,E1 -1206.75,E2 -1206.75} C_VEL
LIN {X 0,Y 594.945,Z 378.575,A -85,B 0,C 180,E1 -1208.311,E2 -1208.311} C_VEL
LIN {X 0,Y 594.411,Z 375.069,A -85,B 0,C 180,E1 -1209.128,E2 -1209.128} C_VEL
LIN {X 0,Y 594.378,Z 375.076,A -85,B 0,C 180,E1 -1211.848,E2 -1211.848} C_VEL
LIN {X 0,Y 594.375,Z 375.07,A -85,B 0,C 180,E1 -1214.235,E2 -1214.235} C_VEL
LIN {X 0,Y 594.378,Z 375.067,A -85,B 0,C 180,E1 -1217.145,E2 -1217.145} C_VEL
LIN {X 0,Y 594.383,Z 375.07,A -85,B 0,C 180,E1 -1219.434,E2 -1219.434} C_VEL
LIN {X 0,Y 594.384,Z 375.066,A -85,B 0,C 180,E1 -1222.39,E2 -1222.39} C_VEL
LIN {X 0,Y 594.375,Z 375.066,A -85,B 0,C 180,E1 -1224.671,E2 -1224.671} C_VEL
LIN {X 0,Y 594.372,Z 375.068,A -85,B 0,C 180,E1 -1227.087,E2 -1227.087} C_VEL
LIN {X 0,Y 594.391,Z 375.075,A -85,B 0,C 180,E1 -1229.669,E2 -1229.669} C_VEL
LIN {X 0,Y 594.381,Z 375.066,A -85,B 0,C 180,E1 -1232.539,E2 -1232.539} C_VEL
LIN {X 0,Y 594.37,Z 375.067,A -85,B 0,C 180,E1 -1234.807,E2 -1234.807} C_VEL
LIN {X 0,Y 594.356,Z 375.073,A -85,B 0,C 180,E1 -1237.263,E2 -1237.263} C_VEL
LIN {X 0,Y 594.371,Z 375.072,A -85,B 0,C 180,E1 -1239.946,E2 -1239.946} C_VEL
LIN {X 0,Y 594.384,Z 375.066,A -85,B 0,C 180,E1 -1242.807,E2 -1242.807} C_VEL
LIN {X 0,Y 594.378,Z 375.072,A -85,B 0,C 180,E1 -1245.825,E2 -1245.825} C_VEL
LIN {X 0,Y 594.385,Z 375.065,A -85,B 0,C 180,E1 -1248.404,E2 -1248.404} C_VEL
LIN {X 0,Y 594.394,Z 375.068,A -85,B 0,C 180,E1 -1251.158,E2 -1251.158} C_VEL
LIN {X 0,Y 594.361,Z 375.072,A -85,B 0,C 180,E1 -1253.891,E2 -1253.891} C_VEL
LIN {X 0,Y 594.379,Z 375.066,A -85,B 0,C 180,E1 -1256.611,E2 -1256.611} C_VEL
LIN {X 0,Y 594.42,Z 375.069,A -85,B 0,C 180,E1 -1259.323,E2 -1259.323} C_VEL
LIN {X 0,Y 594.388,Z 375.067,A -85,B 0,C 180,E1 -1262.033,E2 -1262.033} C_VEL
LIN {X 0,Y 594.395,Z 375.065,A -85,B 0,C 180,E1 -1264.748,E2 -1264.748} C_VEL
LIN {X 0,Y 594.394,Z 375.074,A -85,B 0,C 180,E1 -1267.473,E2 -1267.473} C_VEL
LIN {X 0,Y 594.388,Z 375.065,A -85,B 0,C 180,E1 -1270.216,E2 -1270.216} C_VEL
LIN {X 0,Y 594.366,Z 375.071,A -85,B 0,C 180,E1 -1272.983,E2 -1272.983} C_VEL
LIN {X 0,Y 594.358,Z 375.072,A -85,B 0,C 180,E1 -1275.34,E2 -1275.34} C_VEL
LIN {X 0,Y 593.688,Z 375.155,A -85,B 0,C 180,E1 -1275.906,E2 -1275.906} C_VEL
LIN {X 0,Y 590.834,Z 375.51,A -85,B 0,C 180,E1 -1276.824,E2 -1276.824} C_VEL
LIN {X 0,Y 588.428,Z 375.814,A -85,B 0,C 180,E1 -1277.562,E2 -1277.562} C_VEL
LIN {X 0,Y 587.4,Z 375.936,A -85,B 0,C 180,E1 -1278.133,E2 -1278.133} C_VEL
LIN {X 0,Y 587.319,Z 375.945,A -85,B 0,C 180,E1 -1278.326,E2 -1278.326} C_VEL
LIN {X 0,Y 587.349,Z 375.948,A -85,B 0,C 180,E1 -1281.046,E2 -1281.046} C_VEL
LIN {X 0,Y 587.329,Z 375.945,A -85,B 0,C 180,E1 -1284.007,E2 -1284.007} C_VEL
LIN {X 0,Y 587.356,Z 375.941,A -85,B 0,C 180,E1 -1286.278,E2 -1286.278} C_VEL
LIN {X 0,Y 587.344,Z 375.951,A -85,B 0,C 180,E1 -1289.135,E2 -1289.135} C_VEL
LIN {X 0,Y 587.351,Z 375.943,A -85,B 0,C 180,E1 -1291.839,E2 -1291.839} C_VEL
LIN {X 0,Y 587.348,Z 375.942,A -85,B 0,C 180,E1 -1294.35,E2 -1294.35} C_VEL
LIN {X 0,Y 587.347,Z 375.945,A -85,B 0,C 180,E1 -1296.747,E2 -1296.747} C_VEL
LIN {X 0,Y 587.341,Z 375.95,A -85,B 0,C 180,E1 -1299.36,E2 -1299.36} C_VEL
LIN {X 0,Y 587.332,Z 375.944,A -85,B 0,C 180,E1 -1302.109,E2 -1302.109} C_VEL
LIN {X 0,Y 587.312,Z 375.956,A -85,B 0,C 180,E1 -1305.09,E2 -1305.09} C_VEL
LIN {X 0,Y 587.349,Z 375.942,A -85,B 0,C 180,E1 -1307.929,E2 -1307.929} C_VEL
LIN {X 0,Y 587.334,Z 375.954,A -85,B 0,C 180,E1 -1311.059,E2 -1311.059} C_VEL
LIN {X 0,Y 587.352,Z 375.948,A -85,B 0,C 180,E1 -1313.293,E2 -1313.293} C_VEL
LIN {X 0,Y 587.366,Z 375.94,A -85,B 0,C 180,E1 -1315.782,E2 -1315.782} C_VEL
LIN {X 0,Y 587.351,Z 375.942,A -85,B 0,C 180,E1 -1318.233,E2 -1318.233} C_VEL
LIN {X 0,Y 587.35,Z 375.949,A -85,B 0,C 180,E1 -1320.867,E2 -1320.867} C_VEL
LIN {X 0,Y 587.36,Z 375.941,A -85,B 0,C 180,E1 -1323.82,E2 -1323.82} C_VEL
LIN {X 0,Y 587.337,Z 375.943,A -85,B 0,C 180,E1 -1325.995,E2 -1325.995} C_VEL
LIN {X 0,Y 587.32,Z 375.946,A -85,B 0,C 180,E1 -1328.227,E2 -1328.227} C_VEL
LIN {X 0,Y 587.35,Z 375.949,A -85,B 0,C 180,E1 -1331.152,E2 -1331.152} C_VEL
LIN {X 0,Y 587.321,Z 375.945,A -85,B 0,C 180,E1 -1334.026,E2 -1334.026} C_VEL
LIN {X 0,Y 587.185,Z 375.972,A -85,B 0,C 180,E1 -1336.151,E2 -1336.151} C_VEL
LIN {X 0,Y 587.141,Z 376.383,A -85,B 0,C 180,E1 -1336.855,E2 -1336.855} C_VEL
LIN {X 0,Y 587.134,Z 379.856,A -85,B 0,C 180,E1 -1339.657,E2 -1339.657} C_VEL
LIN {X 0,Y 587.164,Z 381.405,A -85,B 0,C 180,E1 -1340.897,E2 -1340.897} C_VEL
LIN {X 0,Y 587.69,Z 387.179,A -85,B 0,C 180,E1 -1341.036,E2 -1341.036} C_VEL
LIN {X 0,Y 587.666,Z 400.034,A -85,B 0,C 180,E1 -1341.403,E2 -1341.403} C_VEL
LIN {X 0,Y 587.595,Z 410.944,A -85,B 0,C 180,E1 -1341.835,E2 -1341.835} C_VEL
LIN {X 0,Y 587.524,Z 422.69,A -85,B 0,C 180,E1 -1342.44,E2 -1342.44} C_VEL
LIN {X 0,Y 587.418,Z 433.274,A -85,B 0,C 180,E1 -1343.129,E2 -1343.129} C_VEL
LIN {X 0,Y 587.328,Z 443.872,A -85,B 0,C 180,E1 -1343.991,E2 -1343.991} C_VEL
LIN {X 0,Y 587.318,Z 452.497,A -85,B 0,C 180,E1 -1344.852,E2 -1344.852} C_VEL
LIN {X 0,Y 587.288,Z 460.91,A -85,B 0,C 180,E1 -1345.883,E2 -1345.883} C_VEL
LIN {X 0,Y 587.255,Z 467.675,A -85,B 0,C 180,E1 -1346.914,E2 -1346.914} C_VEL
LIN {X 0,Y 587.164,Z 473.096,A -85,B 0,C 180,E1 -1347.943,E2 -1347.943} C_VEL
LIN {X 0,Y 587.167,Z 477.342,A -85,B 0,C 180,E1 -1348.972,E2 -1348.972} C_VEL
LIN {X 0,Y 587.14,Z 480.538,A -85,B 0,C 180,E1 -1350.001,E2 -1350.001} C_VEL
LIN {X 0,Y 587.149,Z 483.318,A -85,B 0,C 180,E1 -1351.372,E2 -1351.372} C_VEL
LIN {X 0,Y 587.14,Z 484.079,A -85,B 0,C 180,E1 -1352.059,E2 -1352.059} C_VEL
LIN {X 0,Y 587.181,Z 484.419,A -85,B 0,C 180,E1 -1353.432,E2 -1353.432} C_VEL
LIN {X 0,Y 587.17,Z 484.014,A -85,B 0,C 180,E1 -1354.119,E2 -1354.119} C_VEL
LIN {X 0,Y 587.179,Z 481.936,A -85,B 0,C 180,E1 -1355.495,E2 -1355.495} C_VEL
LIN {X 0,Y 587.189,Z 479.156,A -85,B 0,C 180,E1 -1356.574,E2 -1356.574} C_VEL
LIN {X 0,Y 587.187,Z 475.631,A -85,B 0,C 180,E1 -1357.566,E2 -1357.566} C_VEL
LIN {X 0,Y 587.214,Z 470.841,A -85,B 0,C 180,E1 -1358.605,E2 -1358.605} C_VEL
LIN {X 0,Y 587.248,Z 464.773,A -85,B 0,C 180,E1 -1359.646,E2 -1359.646} C_VEL
LIN {X 0,Y 587.269,Z 457.202,A -85,B 0,C 180,E1 -1360.69,E2 -1360.69} C_VEL
LIN {X 0,Y 587.317,Z 449.622,A -85,B 0,C 180,E1 -1361.546,E2 -1361.546} C_VEL
LIN {X 0,Y 587.359,Z 439.971,A -85,B 0,C 180,E1 -1362.438,E2 -1362.438} C_VEL
LIN {X 0,Y 587.477,Z 429.438,A -85,B 0,C 180,E1 -1363.227,E2 -1363.227} C_VEL
LIN {X 0,Y 587.529,Z 419.272,A -85,B 0,C 180,E1 -1363.842,E2 -1363.842} C_VEL
LIN {X 0,Y 587.604,Z 407.74,A -85,B 0,C 180,E1 -1364.395,E2 -1364.395} C_VEL
LIN {X 0,Y 587.672,Z 394.755,A -85,B 0,C 180,E1 -1364.856,E2 -1364.856} C_VEL
LIN {X 0,Y 587.556,Z 384.088,A -85,B 0,C 180,E1 -1365.125,E2 -1365.125} C_VEL
LIN {X 0,Y 587.17,Z 381.394,A -85,B 0,C 180,E1 -1365.201,E2 -1365.201} C_VEL
LIN {X 0,Y 587.125,Z 377.743,A -85,B 0,C 180,E1 -1368.134,E2 -1368.134} C_VEL
LIN {X 0,Y 587.118,Z 375.977,A -85,B 0,C 180,E1 -1369.583,E2 -1369.583} C_VEL
LIN {X 0,Y 587.318,Z 375.947,A -85,B 0,C 180,E1 -1371.775,E2 -1371.775} C_VEL
LIN {X 0,Y 587.358,Z 375.946,A -85,B 0,C 180,E1 -1374.759,E2 -1374.759} C_VEL
LIN {X 0,Y 587.348,Z 375.943,A -85,B 0,C 180,E1 -1377.691,E2 -1377.691} C_VEL
LIN {X 0,Y 587.342,Z 375.948,A -85,B 0,C 180,E1 -1380.51,E2 -1380.51} C_VEL
LIN {X 0,Y 587.333,Z 375.946,A -85,B 0,C 180,E1 -1383.397,E2 -1383.397} C_VEL
LIN {X 0,Y 587.298,Z 375.949,A -85,B 0,C 180,E1 -1385.9,E2 -1385.9} C_VEL
LIN {X 0,Y 587.334,Z 375.951,A -85,B 0,C 180,E1 -1388.48,E2 -1388.48} C_VEL
LIN {X 0,Y 587.339,Z 375.944,A -85,B 0,C 180,E1 -1391.157,E2 -1391.157} C_VEL
LIN {X 0,Y 587.332,Z 375.949,A -85,B 0,C 180,E1 -1394.113,E2 -1394.113} C_VEL
LIN {X 0,Y 587.326,Z 375.946,A -85,B 0,C 180,E1 -1396.994,E2 -1396.994} C_VEL
LIN {X 0,Y 587.322,Z 375.947,A -85,B 0,C 180,E1 -1399.746,E2 -1399.746} C_VEL
LIN {X 0,Y 587.35,Z 375.946,A -85,B 0,C 180,E1 -1402.392,E2 -1402.392} C_VEL
LIN {X 0,Y 587.328,Z 375.944,A -85,B 0,C 180,E1 -1404.944,E2 -1404.944} C_VEL
LIN {X 0,Y 587.341,Z 375.945,A -85,B 0,C 180,E1 -1407.421,E2 -1407.421} C_VEL
LIN {X 0,Y 587.337,Z 375.95,A -85,B 0,C 180,E1 -1409.83,E2 -1409.83} C_VEL
LIN {X 0,Y 587.355,Z 375.942,A -85,B 0,C 180,E1 -1412.307,E2 -1412.307} C_VEL
LIN {X 0,Y 587.353,Z 375.944,A -85,B 0,C 180,E1 -1415.241,E2 -1415.241} C_VEL
LIN {X 0,Y 587.326,Z 375.946,A -85,B 0,C 180,E1 -1418.226,E2 -1418.226} C_VEL
LIN {X 0,Y 587.352,Z 375.946,A -85,B 0,C 180,E1 -1421.151,E2 -1421.151} C_VEL
LIN {X 0,Y 587.325,Z 375.947,A -85,B 0,C 180,E1 -1424.025,E2 -1424.025} C_VEL
LIN {X 0,Y 587.364,Z 375.944,A -85,B 0,C 180,E1 -1426.793,E2 -1426.793} C_VEL
LIN {X 0,Y 587.909,Z 379.209,A -85,B 0,C 180,E1 -1426.916,E2 -1426.916} C_VEL
LIN {X 0,Y 587.826,Z 392.389,A -85,B 0,C 180,E1 -1427.397,E2 -1427.397} C_VEL
LIN {X 0,Y 587.686,Z 405.204,A -85,B 0,C 180,E1 -1428.007,E2 -1428.007} C_VEL
LIN {X 0,Y 587.571,Z 417.69,A -85,B 0,C 180,E1 -1428.758,E2 -1428.758} C_VEL
LIN {X 0,Y 587.494,Z 428.847,A -85,B 0,C 180,E1 -1429.576,E2 -1429.576} C_VEL
LIN {X 0,Y 587.413,Z 439.616,A -85,B 0,C 180,E1 -1430.531,E2 -1430.531} C_VEL
LIN {X 0,Y 587.34,Z 449.314,A -85,B 0,C 180,E1 -1431.571,E2 -1431.571} C_VEL
LIN {X 0,Y 587.271,Z 457.357,A -85,B 0,C 180,E1 -1432.608,E2 -1432.608} C_VEL
LIN {X 0,Y 587.222,Z 465.065,A -85,B 0,C 180,E1 -1433.816,E2 -1433.816} C_VEL
LIN {X 0,Y 587.168,Z 470.476,A -85,B 0,C 180,E1 -1434.849,E2 -1434.849} C_VEL
LIN {X 0,Y 587.211,Z 476.158,A -85,B 0,C 180,E1 -1436.226,E2 -1436.226} C_VEL
LIN {X 0,Y 587.138,Z 479.396,A -85,B 0,C 180,E1 -1437.255,E2 -1437.255} C_VEL
LIN {X 0,Y 587.142,Z 482.415,A -85,B 0,C 180,E1 -1438.628,E2 -1438.628} C_VEL
LIN {X 0,Y 587.135,Z 484.083,A -85,B 0,C 180,E1 -1440,E2 -1440} C_VEL
LIN {X 0,Y 587.146,Z 484.436,A -85,B 0,C 180,E1 -1441.372,E2 -1441.372} C_VEL
LIN {X 0,Y 587.128,Z 483.467,A -85,B 0,C 180,E1 -1442.744,E2 -1442.744} C_VEL
LIN {X 0,Y 587.168,Z 481.15,A -85,B 0,C 180,E1 -1444.118,E2 -1444.118} C_VEL
LIN {X 0,Y 587.193,Z 477.407,A -85,B 0,C 180,E1 -1445.494,E2 -1445.494} C_VEL
LIN {X 0,Y 587.208,Z 472.18,A -85,B 0,C 180,E1 -1446.874,E2 -1446.874} C_VEL
LIN {X 0,Y 587.218,Z 467.101,A -85,B 0,C 180,E1 -1447.911,E2 -1447.911} C_VEL
LIN {X 0,Y 587.268,Z 459.839,A -85,B 0,C 180,E1 -1449.124,E2 -1449.124} C_VEL
LIN {X 0,Y 587.3,Z 452.212,A -85,B 0,C 180,E1 -1450.166,E2 -1450.166} C_VEL
LIN {X 0,Y 587.379,Z 442.559,A -85,B 0,C 180,E1 -1451.263,E2 -1451.263} C_VEL
LIN {X 0,Y 587.473,Z 431.946,A -85,B 0,C 180,E1 -1452.26,E2 -1452.26} C_VEL
LIN {X 0,Y 587.586,Z 420.559,A -85,B 0,C 180,E1 -1453.135,E2 -1453.135} C_VEL
LIN {X 0,Y 587.66,Z 408.549,A -85,B 0,C 180,E1 -1453.895,E2 -1453.895} C_VEL
LIN {X 0,Y 587.788,Z 395.835,A -85,B 0,C 180,E1 -1454.542,E2 -1454.542} C_VEL
LIN {X 0,Y 587.89,Z 381.1,A -85,B 0,C 180,E1 -1455.115,E2 -1455.115} C_VEL
LIN {X 0,Y 587.716,Z 377.46,A -85,B 0,C 180,E1 -1455.233,E2 -1455.233} C_VEL
LIN {X 0,Y 587.34,Z 375.953,A -85,B 0,C 180,E1 -1455.307,E2 -1455.307} C_VEL
LIN {X 0,Y 587.362,Z 375.947,A -85,B 0,C 180,E1 -1457.405,E2 -1457.405} C_VEL
LIN {X 0,Y 587.331,Z 375.954,A -85,B 0,C 180,E1 -1460.305,E2 -1460.305} C_VEL
LIN {X 0,Y 587.328,Z 375.951,A -85,B 0,C 180,E1 -1463.258,E2 -1463.258} C_VEL
LIN {X 0,Y 587.333,Z 375.952,A -85,B 0,C 180,E1 -1465.517,E2 -1465.517} C_VEL
LIN {X 0,Y 587.352,Z 375.952,A -85,B 0,C 180,E1 -1467.817,E2 -1467.817} C_VEL
LIN {X 0,Y 587.338,Z 375.951,A -85,B 0,C 180,E1 -1470.51,E2 -1470.51} C_VEL
LIN {X 0,Y 587.339,Z 375.949,A -85,B 0,C 180,E1 -1473.396,E2 -1473.396} C_VEL
LIN {X 0,Y 587.293,Z 375.955,A -85,B 0,C 180,E1 -1475.9,E2 -1475.9} C_VEL
LIN {X 0,Y 587.334,Z 375.95,A -85,B 0,C 180,E1 -1478.479,E2 -1478.479} C_VEL
LIN {X 0,Y 587.339,Z 375.95,A -85,B 0,C 180,E1 -1481.157,E2 -1481.157} C_VEL
LIN {X 0,Y 587.338,Z 375.953,A -85,B 0,C 180,E1 -1484.114,E2 -1484.114} C_VEL
LIN {X 0,Y 587.318,Z 375.953,A -85,B 0,C 180,E1 -1486.993,E2 -1486.993} C_VEL
LIN {X 0,Y 587.319,Z 375.952,A -85,B 0,C 180,E1 -1489.746,E2 -1489.746} C_VEL
LIN {X 0,Y 587.36,Z 375.966,A -85,B 0,C 180,E1 -1491.817,E2 -1491.817} C_VEL
LIN {X 0,Y 587.551,Z 382.462,A -85,B 0,C 180,E1 -1493.053,E2 -1493.053} C_VEL
LIN {X 0,Y 587.518,Z 399.893,A -85,B 0,C 180,E1 -1496.203,E2 -1496.203} C_VEL
LIN {X 0,Y 587.842,Z 413.901,A -85,B 0,C 180,E1 -1498.663,E2 -1498.663} C_VEL
LIN {X 0,Y 587.966,Z 420.606,A -85,B 0,C 180,E1 -1499.865,E2 -1499.865} C_VEL
LIN {X 0,Y 587.827,Z 434.045,A -85,B 0,C 180,E1 -1502.599,E2 -1502.599} C_VEL
LIN {X 0,Y 587.706,Z 447.849,A -85,B 0,C 180,E1 -1505.345,E2 -1505.345} C_VEL
LIN {X 0,Y 587.571,Z 462.702,A -85,B 0,C 180,E1 -1508.235,E2 -1508.235} C_VEL
LIN {X 0,Y 587.481,Z 478.001,A -85,B 0,C 180,E1 -1511.155,E2 -1511.155} C_VEL
LIN {X 0,Y 587.356,Z 493.301,A -85,B 0,C 180,E1 -1514.025,E2 -1514.025} C_VEL
LIN {X 0,Y 587.364,Z 499.756,A -85,B 0,C 180,E1 -1515.225,E2 -1515.225} C_VEL
LIN {X 0,Y 588.018,Z 504.077,A -85,B 0,C 180,E1 -1515.308,E2 -1515.308} C_VEL
LIN {X 0,Y 587.94,Z 518.221,A -85,B 0,C 180,E1 -1515.569,E2 -1515.569} C_VEL
LIN {X 0,Y 587.883,Z 532.537,A -85,B 0,C 180,E1 -1515.98,E2 -1515.98} C_VEL
LIN {X 0,Y 587.785,Z 546.116,A -85,B 0,C 180,E1 -1516.516,E2 -1516.516} C_VEL
LIN {X 0,Y 587.639,Z 558.202,A -85,B 0,C 180,E1 -1517.129,E2 -1517.129} C_VEL
LIN {X 0,Y 587.588,Z 570.697,A -85,B 0,C 180,E1 -1517.917,E2 -1517.917} C_VEL
LIN {X 0,Y 587.463,Z 582.254,A -85,B 0,C 180,E1 -1518.811,E2 -1518.811} C_VEL
LIN {X 0,Y 587.376,Z 593.075,A -85,B 0,C 180,E1 -1519.834,E2 -1519.834} C_VEL
LIN {X 0,Y 587.322,Z 602.194,A -85,B 0,C 180,E1 -1520.877,E2 -1520.877} C_VEL
LIN {X 0,Y 587.261,Z 610.915,A -85,B 0,C 180,E1 -1522.089,E2 -1522.089} C_VEL
LIN {X 0,Y 587.209,Z 618.523,A -85,B 0,C 180,E1 -1523.406,E2 -1523.406} C_VEL
LIN {X 0,Y 587.199,Z 623.565,A -85,B 0,C 180,E1 -1524.505,E2 -1524.505} C_VEL
LIN {X 0,Y 587.179,Z 628.441,A -85,B 0,C 180,E1 -1525.881,E2 -1525.881} C_VEL
LIN {X 0,Y 587.13,Z 631.831,A -85,B 0,C 180,E1 -1527.255,E2 -1527.255} C_VEL
LIN {X 0,Y 587.141,Z 633.831,A -85,B 0,C 180,E1 -1528.627,E2 -1528.627} C_VEL
LIN {X 0,Y 587.135,Z 634.5,A -85,B 0,C 180,E1 -1529.999,E2 -1529.999} C_VEL
LIN {X 0,Y 587.141,Z 633.832,A -85,B 0,C 180,E1 -1531.371,E2 -1531.371} C_VEL
LIN {X 0,Y 587.13,Z 631.833,A -85,B 0,C 180,E1 -1532.744,E2 -1532.744} C_VEL
LIN {X 0,Y 587.179,Z 628.444,A -85,B 0,C 180,E1 -1534.117,E2 -1534.117} C_VEL
LIN {X 0,Y 587.199,Z 623.571,A -85,B 0,C 180,E1 -1535.494,E2 -1535.494} C_VEL
LIN {X 0,Y 587.208,Z 617.056,A -85,B 0,C 180,E1 -1536.873,E2 -1536.873} C_VEL
LIN {X 0,Y 587.268,Z 609.804,A -85,B 0,C 180,E1 -1538.083,E2 -1538.083} C_VEL
LIN {X 0,Y 587.33,Z 600.83,A -85,B 0,C 180,E1 -1539.296,E2 -1539.296} C_VEL
LIN {X 0,Y 587.371,Z 591.4,A -85,B 0,C 180,E1 -1540.338,E2 -1540.338} C_VEL
LIN {X 0,Y 587.474,Z 581.034,A -85,B 0,C 180,E1 -1541.29,E2 -1541.29} C_VEL
LIN {X 0,Y 587.577,Z 569.442,A -85,B 0,C 180,E1 -1542.169,E2 -1542.169} C_VEL
LIN {X 0,Y 587.667,Z 556.662,A -85,B 0,C 180,E1 -1542.957,E2 -1542.957} C_VEL
LIN {X 0,Y 587.795,Z 544.182,A -85,B 0,C 180,E1 -1543.57,E2 -1543.57} C_VEL
LIN {X 0,Y 587.893,Z 530.747,A -85,B 0,C 180,E1 -1544.081,E2 -1544.081} C_VEL
LIN {X 0,Y 587.942,Z 517.043,A -85,B 0,C 180,E1 -1544.46,E2 -1544.46} C_VEL
LIN {X 0,Y 587.869,Z 502.67,A -85,B 0,C 180,E1 -1544.716,E2 -1544.716} C_VEL
LIN {X 0,Y 587.36,Z 499.764,A -85,B 0,C 180,E1 -1544.773,E2 -1544.773} C_VEL
LIN {X 0,Y 587.457,Z 483.747,A -85,B 0,C 180,E1 -1547.761,E2 -1547.761} C_VEL
LIN {X 0,Y 587.536,Z 468.447,A -85,B 0,C 180,E1 -1550.662,E2 -1550.662} C_VEL
LIN {X 0,Y 587.642,Z 455.06,A -85,B 0,C 180,E1 -1553.244,E2 -1553.244} C_VEL
LIN {X 0,Y 587.756,Z 441.673,A -85,B 0,C 180,E1 -1555.876,E2 -1555.876} C_VEL
LIN {X 0,Y 587.863,Z 428.285,A -85,B 0,C 180,E1 -1558.567,E2 -1558.567} C_VEL
LIN {X 0,Y 587.933,Z 418.176,A -85,B 0,C 180,E1 -1560.608,E2 -1560.608} C_VEL
LIN {X 0,Y 587.885,Z 404.182,A -85,B 0,C 180,E1 -1563.36,E2 -1563.36} C_VEL
LIN {X 0,Y 587.988,Z 389.134,A -85,B 0,C 180,E1 -1566.486,E2 -1566.486} C_VEL
LIN {X 0,Y 588.066,Z 380.081,A -85,B 0,C 180,E1 -1568.421,E2 -1568.421} C_VEL
LIN {X 0,Y 587.351,Z 375.95,A -85,B 0,C 180,E1 -1569.413,E2 -1569.413} C_VEL
LIN {X 0,Y 587.328,Z 375.95,A -85,B 0,C 180,E1 -1572.107,E2 -1572.107} C_VEL
LIN {X 0,Y 587.309,Z 375.948,A -85,B 0,C 180,E1 -1575.088,E2 -1575.088} C_VEL
LIN {X 0,Y 587.345,Z 375.95,A -85,B 0,C 180,E1 -1577.927,E2 -1577.927} C_VEL
LIN {X 0,Y 587.339,Z 375.943,A -85,B 0,C 180,E1 -1580.64,E2 -1580.64} C_VEL
LIN {X 0,Y 587.346,Z 375.945,A -85,B 0,C 180,E1 -1583.291,E2 -1583.291} C_VEL
LIN {X 0,Y 587.359,Z 375.95,A -85,B 0,C 180,E1 -1585.78,E2 -1585.78} C_VEL
LIN {X 0,Y 587.347,Z 375.944,A -85,B 0,C 180,E1 -1588.232,E2 -1588.232} C_VEL
LIN {X 0,Y 587.344,Z 375.943,A -85,B 0,C 180,E1 -1590.865,E2 -1590.865} C_VEL
LIN {X 0,Y 587.353,Z 375.949,A -85,B 0,C 180,E1 -1593.817,E2 -1593.817} C_VEL
LIN {X 0,Y 587.328,Z 375.949,A -85,B 0,C 180,E1 -1595.993,E2 -1595.993} C_VEL
LIN {X 0,Y 587.337,Z 375.944,A -85,B 0,C 180,E1 -1598.963,E2 -1598.963} C_VEL
LIN {X 0,Y 587.322,Z 375.951,A -85,B 0,C 180,E1 -1601.873,E2 -1601.873} C_VEL
LIN {X 0,Y 587.322,Z 375.948,A -85,B 0,C 180,E1 -1604.025,E2 -1604.025} C_VEL
LIN {X 0,Y 587.351,Z 375.943,A -85,B 0,C 180,E1 -1606.154,E2 -1606.154} C_VEL
LIN {X 0,Y 587.337,Z 375.945,A -85,B 0,C 180,E1 -1608.962,E2 -1608.962} C_VEL
LIN {X 0,Y 587.363,Z 375.947,A -85,B 0,C 180,E1 -1611.745,E2 -1611.745} C_VEL
LIN {X 0,Y 587.352,Z 375.941,A -85,B 0,C 180,E1 -1614.507,E2 -1614.507} C_VEL
LIN {X 0,Y 587.375,Z 375.945,A -85,B 0,C 180,E1 -1617.257,E2 -1617.257} C_VEL
LIN {X 0,Y 587.373,Z 375.941,A -85,B 0,C 180,E1 -1620,E2 -1620} C_VEL
LIN {X 0,Y 587.373,Z 375.94,A -85,B 0,C 180,E1 -1622.743,E2 -1622.743} C_VEL
LIN {X 0,Y 587.353,Z 375.95,A -85,B 0,C 180,E1 -1625.493,E2 -1625.493} C_VEL
LIN {X 0,Y 587.363,Z 375.94,A -85,B 0,C 180,E1 -1628.256,E2 -1628.256} C_VEL
LIN {X 0,Y 587.352,Z 375.948,A -85,B 0,C 180,E1 -1631.142,E2 -1631.142} C_VEL
LIN {X 0,Y 587.355,Z 375.941,A -85,B 0,C 180,E1 -1634.261,E2 -1634.261} C_VEL
LIN {X 0,Y 587.353,Z 375.95,A -85,B 0,C 180,E1 -1637.406,E2 -1637.406} C_VEL
LIN {X 0,Y 587.319,Z 375.945,A -85,B 0,C 180,E1 -1638.326,E2 -1638.326} C_VEL
LIN {X 0,Y 586.666,Z 376.031,A -85,B 0,C 180,E1 -1638.898,E2 -1638.898} C_VEL
LIN {X 0,Y 583.836,Z 376.392,A -85,B 0,C 180,E1 -1639.826,E2 -1639.826} C_VEL
LIN {X 0,Y 581.427,Z 376.695,A -85,B 0,C 180,E1 -1640.573,E2 -1640.573} C_VEL
LIN {X 0,Y 580.375,Z 376.823,A -85,B 0,C 180,E1 -1641.149,E2 -1641.149} C_VEL
LIN {X 0,Y 580.28,Z 376.831,A -85,B 0,C 180,E1 -1641.344,E2 -1641.344} C_VEL
LIN {X 0,Y 580.293,Z 376.821,A -85,B 0,C 180,E1 -1644.317,E2 -1644.317} C_VEL
LIN {X 0,Y 580.303,Z 376.821,A -85,B 0,C 180,E1 -1646.622,E2 -1646.622} C_VEL
LIN {X 0,Y 580.296,Z 376.829,A -85,B 0,C 180,E1 -1649.311,E2 -1649.311} C_VEL
LIN {X 0,Y 580.298,Z 376.82,A -85,B 0,C 180,E1 -1652.201,E2 -1652.201} C_VEL
LIN {X 0,Y 580.294,Z 376.823,A -85,B 0,C 180,E1 -1654.696,E2 -1654.696} C_VEL
LIN {X 0,Y 580.295,Z 376.829,A -85,B 0,C 180,E1 -1657.269,E2 -1657.269} C_VEL
LIN {X 0,Y 580.294,Z 376.821,A -85,B 0,C 180,E1 -1660.273,E2 -1660.273} C_VEL
LIN {X 0,Y 580.286,Z 376.825,A -85,B 0,C 180,E1 -1662.706,E2 -1662.706} C_VEL
LIN {X 0,Y 580.27,Z 376.827,A -85,B 0,C 180,E1 -1665.61,E2 -1665.61} C_VEL
LIN {X 0,Y 580.31,Z 376.819,A -85,B 0,C 180,E1 -1668.235,E2 -1668.235} C_VEL
LIN {X 0,Y 580.289,Z 376.829,A -85,B 0,C 180,E1 -1670.967,E2 -1670.967} C_VEL
LIN {X 0,Y 580.295,Z 376.823,A -85,B 0,C 180,E1 -1673.6,E2 -1673.6} C_VEL
LIN {X 0,Y 580.318,Z 376.818,A -85,B 0,C 180,E1 -1676.147,E2 -1676.147} C_VEL
LIN {X 0,Y 580.287,Z 376.825,A -85,B 0,C 180,E1 -1678.616,E2 -1678.616} C_VEL
LIN {X 0,Y 580.292,Z 376.83,A -85,B 0,C 180,E1 -1681.025,E2 -1681.025} C_VEL
LIN {X 0,Y 580.292,Z 376.822,A -85,B 0,C 180,E1 -1683.667,E2 -1683.667} C_VEL
LIN {X 0,Y 580.301,Z 376.821,A -85,B 0,C 180,E1 -1685.685,E2 -1685.685} C_VEL
LIN {X 0,Y 580.271,Z 376.824,A -85,B 0,C 180,E1 -1687.948,E2 -1687.948} C_VEL
LIN {X 0,Y 580.3,Z 376.83,A -85,B 0,C 180,E1 -1690.914,E2 -1690.914} C_VEL
LIN {X 0,Y 580.271,Z 376.824,A -85,B 0,C 180,E1 -1693.826,E2 -1693.826} C_VEL
LIN {X 0,Y 580.154,Z 376.846,A -85,B 0,C 180,E1 -1695.98,E2 -1695.98} C_VEL
LIN {X 0,Y 580.094,Z 376.852,A -85,B 0,C 180,E1 -1696.693,E2 -1696.693} C_VEL
LIN {X 0,Y 580.075,Z 377.298,A -85,B 0,C 180,E1 -1697.405,E2 -1697.405} C_VEL
LIN {X 0,Y 580.049,Z 380.773,A -85,B 0,C 180,E1 -1700.235,E2 -1700.235} C_VEL
LIN {X 0,Y 580.083,Z 381.398,A -85,B 0,C 180,E1 -1700.741,E2 -1700.741} C_VEL
LIN {X 0,Y 580.748,Z 386.931,A -85,B 0,C 180,E1 -1700.884,E2 -1700.884} C_VEL
LIN {X 0,Y 580.713,Z 399.859,A -85,B 0,C 180,E1 -1701.256,E2 -1701.256} C_VEL
LIN {X 0,Y 580.619,Z 411.765,A -85,B 0,C 180,E1 -1701.737,E2 -1701.737} C_VEL
LIN {X 0,Y 580.529,Z 423.332,A -85,B 0,C 180,E1 -1702.348,E2 -1702.348} C_VEL
LIN {X 0,Y 580.401,Z 433.772,A -85,B 0,C 180,E1 -1703.046,E2 -1703.046} C_VEL
LIN {X 0,Y 580.279,Z 444.283,A -85,B 0,C 180,E1 -1703.917,E2 -1703.917} C_VEL
LIN {X 0,Y 580.273,Z 452.834,A -85,B 0,C 180,E1 -1704.789,E2 -1704.789} C_VEL
LIN {X 0,Y 580.22,Z 461.176,A -85,B 0,C 180,E1 -1705.833,E2 -1705.833} C_VEL
LIN {X 0,Y 580.194,Z 467.892,A -85,B 0,C 180,E1 -1706.876,E2 -1706.876} C_VEL
LIN {X 0,Y 580.07,Z 473.271,A -85,B 0,C 180,E1 -1707.918,E2 -1707.918} C_VEL
LIN {X 0,Y 580.087,Z 477.475,A -85,B 0,C 180,E1 -1708.959,E2 -1708.959} C_VEL
LIN {X 0,Y 580.041,Z 480.633,A -85,B 0,C 180,E1 -1710.001,E2 -1710.001} C_VEL
LIN {X 0,Y 580.04,Z 482.204,A -85,B 0,C 180,E1 -1710.695,E2 -1710.695} C_VEL
LIN {X 0,Y 580.049,Z 483.373,A -85,B 0,C 180,E1 -1711.389,E2 -1711.389} C_VEL
LIN {X 0,Y 580.039,Z 484.447,A -85,B 0,C 180,E1 -1712.779,E2 -1712.779} C_VEL
LIN {X 0,Y 580.107,Z 484.41,A -85,B 0,C 180,E1 -1713.474,E2 -1713.474} C_VEL
LIN {X 0,Y 580.088,Z 483.979,A -85,B 0,C 180,E1 -1714.169,E2 -1714.169} C_VEL
LIN {X 0,Y 580.099,Z 481.859,A -85,B 0,C 180,E1 -1715.563,E2 -1715.563} C_VEL
LIN {X 0,Y 580.1,Z 479.324,A -85,B 0,C 180,E1 -1716.562,E2 -1716.562} C_VEL
LIN {X 0,Y 580.107,Z 475.478,A -85,B 0,C 180,E1 -1717.659,E2 -1717.659} C_VEL
LIN {X 0,Y 580.117,Z 470.646,A -85,B 0,C 180,E1 -1718.711,E2 -1718.711} C_VEL
LIN {X 0,Y 580.196,Z 464.533,A -85,B 0,C 180,E1 -1719.764,E2 -1719.764} C_VEL
LIN {X 0,Y 580.219,Z 457.217,A -85,B 0,C 180,E1 -1720.782,E2 -1720.782} C_VEL
LIN {X 0,Y 580.283,Z 449.074,A -85,B 0,C 180,E1 -1721.705,E2 -1721.705} C_VEL
LIN {X 0,Y 580.354,Z 439.513,A -85,B 0,C 180,E1 -1722.591,E2 -1722.591} C_VEL
LIN {X 0,Y 580.463,Z 428.884,A -85,B 0,C 180,E1 -1723.389,E2 -1723.389} C_VEL
LIN {X 0,Y 580.541,Z 418.589,A -85,B 0,C 180,E1 -1724.012,E2 -1724.012} C_VEL
LIN {X 0,Y 580.658,Z 405.885,A -85,B 0,C 180,E1 -1724.609,E2 -1724.609} C_VEL
LIN {X 0,Y 580.713,Z 392.67,A -85,B 0,C 180,E1 -1725.06,E2 -1725.06} C_VEL
LIN {X 0,Y 580.565,Z 384.647,A -85,B 0,C 180,E1 -1725.261,E2 -1725.261} C_VEL
LIN {X 0,Y 580.068,Z 381.401,A -85,B 0,C 180,E1 -1725.347,E2 -1725.347} C_VEL
LIN {X 0,Y 580.034,Z 377.693,A -85,B 0,C 180,E1 -1728.363,E2 -1728.363} C_VEL
LIN {X 0,Y 580.063,Z 376.855,A -85,B 0,C 180,E1 -1729.095,E2 -1729.095} C_VEL
LIN {X 0,Y 580.272,Z 376.831,A -85,B 0,C 180,E1 -1731.306,E2 -1731.306} C_VEL
LIN {X 0,Y 580.278,Z 376.826,A -85,B 0,C 180,E1 -1733.559,E2 -1733.559} C_VEL
LIN {X 0,Y 580.288,Z 376.822,A -85,B 0,C 180,E1 -1735.85,E2 -1735.85} C_VEL
LIN {X 0,Y 580.301,Z 376.821,A -85,B 0,C 180,E1 -1738.186,E2 -1738.186} C_VEL
LIN {X 0,Y 580.289,Z 376.829,A -85,B 0,C 180,E1 -1740.694,E2 -1740.694} C_VEL
LIN {X 0,Y 580.288,Z 376.824,A -85,B 0,C 180,E1 -1743.313,E2 -1743.313} C_VEL
LIN {X 0,Y 580.253,Z 376.826,A -85,B 0,C 180,E1 -1745.757,E2 -1745.757} C_VEL
LIN {X 0,Y 580.293,Z 376.823,A -85,B 0,C 180,E1 -1748.146,E2 -1748.146} C_VEL
LIN {X 0,Y 580.302,Z 376.824,A -85,B 0,C 180,E1 -1750.844,E2 -1750.844} C_VEL
LIN {X 0,Y 580.284,Z 376.823,A -85,B 0,C 180,E1 -1753.658,E2 -1753.658} C_VEL
LIN {X 0,Y 580.291,Z 376.826,A -85,B 0,C 180,E1 -1756.608,E2 -1756.608} C_VEL
LIN {X 0,Y 580.304,Z 376.819,A -85,B 0,C 180,E1 -1759.157,E2 -1759.157} C_VEL
LIN {X 0,Y 580.296,Z 376.823,A -85,B 0,C 180,E1 -1761.927,E2 -1761.927} C_VEL
LIN {X 0,Y 580.289,Z 376.825,A -85,B 0,C 180,E1 -1764.455,E2 -1764.455} C_VEL
LIN {X 0,Y 580.294,Z 376.82,A -85,B 0,C 180,E1 -1766.975,E2 -1766.975} C_VEL
LIN {X 0,Y 580.299,Z 376.82,A -85,B 0,C 180,E1 -1769.425,E2 -1769.425} C_VEL
LIN {X 0,Y 580.301,Z 376.823,A -85,B 0,C 180,E1 -1772.141,E2 -1772.141} C_VEL
LIN {X 0,Y 580.324,Z 376.82,A -85,B 0,C 180,E1 -1775.27,E2 -1775.27} C_VEL
LIN {X 0,Y 580.276,Z 376.828,A -85,B 0,C 180,E1 -1777.947,E2 -1777.947} C_VEL
LIN {X 0,Y 580.302,Z 376.822,A -85,B 0,C 180,E1 -1780.913,E2 -1780.913} C_VEL
LIN {X 0,Y 580.28,Z 376.827,A -85,B 0,C 180,E1 -1783.825,E2 -1783.825} C_VEL
LIN {X 0,Y 580.326,Z 376.82,A -85,B 0,C 180,E1 -1786.652,E2 -1786.652} C_VEL
LIN {X 0,Y 581.018,Z 379.602,A -85,B 0,C 180,E1 -1786.758,E2 -1786.758} C_VEL
LIN {X 0,Y 580.92,Z 392.699,A -85,B 0,C 180,E1 -1787.244,E2 -1787.244} C_VEL
LIN {X 0,Y 580.735,Z 405.434,A -85,B 0,C 180,E1 -1787.862,E2 -1787.862} C_VEL
LIN {X 0,Y 580.623,Z 417.152,A -85,B 0,C 180,E1 -1788.572,E2 -1788.572} C_VEL
LIN {X 0,Y 580.53,Z 427.899,A -85,B 0,C 180,E1 -1789.361,E2 -1789.361} C_VEL
LIN {X 0,Y 580.358,Z 437.941,A -85,B 0,C 180,E1 -1790.239,E2 -1790.239} C_VEL
LIN {X 0,Y 580.274,Z 447.943,A -85,B 0,C 180,E1 -1791.292,E2 -1791.292} C_VEL
LIN {X 0,Y 580.226,Z 457.448,A -85,B 0,C 180,E1 -1792.518,E2 -1792.518} C_VEL
LIN {X 0,Y 580.149,Z 464.342,A -85,B 0,C 180,E1 -1793.603,E2 -1793.603} C_VEL
LIN {X 0,Y 580.086,Z 470.536,A -85,B 0,C 180,E1 -1794.786,E2 -1794.786} C_VEL
LIN {X 0,Y 580.138,Z 476.207,A -85,B 0,C 180,E1 -1796.179,E2 -1796.179} C_VEL
LIN {X 0,Y 580.049,Z 479.431,A -85,B 0,C 180,E1 -1797.222,E2 -1797.222} C_VEL
LIN {X 0,Y 580.042,Z 482.433,A -85,B 0,C 180,E1 -1798.611,E2 -1798.611} C_VEL
LIN {X 0,Y 580.035,Z 484.09,A -85,B 0,C 180,E1 -1800,E2 -1800} C_VEL
LIN {X 0,Y 580.046,Z 484.435,A -85,B 0,C 180,E1 -1801.388,E2 -1801.388} C_VEL
LIN {X 0,Y 580.039,Z 483.455,A -85,B 0,C 180,E1 -1802.778,E2 -1802.778} C_VEL
LIN {X 0,Y 580.086,Z 481.124,A -85,B 0,C 180,E1 -1804.168,E2 -1804.168} C_VEL
LIN {X 0,Y 580.117,Z 477.361,A -85,B 0,C 180,E1 -1805.562,E2 -1805.562} C_VEL
LIN {X 0,Y 580.139,Z 472.124,A -85,B 0,C 180,E1 -1806.958,E2 -1806.958} C_VEL
LIN {X 0,Y 580.151,Z 467.037,A -85,B 0,C 180,E1 -1808.008,E2 -1808.008} C_VEL
LIN {X 0,Y 580.211,Z 459.752,A -85,B 0,C 180,E1 -1809.235,E2 -1809.235} C_VEL
LIN {X 0,Y 580.267,Z 452.1,A -85,B 0,C 180,E1 -1810.291,E2 -1810.291} C_VEL
LIN {X 0,Y 580.348,Z 443.082,A -85,B 0,C 180,E1 -1811.331,E2 -1811.331} C_VEL
LIN {X 0,Y 580.44,Z 431.789,A -85,B 0,C 180,E1 -1812.411,E2 -1812.411} C_VEL
LIN {X 0,Y 580.605,Z 420.363,A -85,B 0,C 180,E1 -1813.296,E2 -1813.296} C_VEL
LIN {X 0,Y 580.711,Z 409.298,A -85,B 0,C 180,E1 -1814.007,E2 -1814.007} C_VEL
LIN {X 0,Y 580.872,Z 396.641,A -85,B 0,C 180,E1 -1814.669,E2 -1814.669} C_VEL
LIN {X 0,Y 581.005,Z 382.026,A -85,B 0,C 180,E1 -1815.254,E2 -1815.254} C_VEL
LIN {X 0,Y 580.783,Z 378.621,A -85,B 0,C 180,E1 -1815.369,E2 -1815.369} C_VEL
LIN {X 0,Y 580.334,Z 376.825,A -85,B 0,C 180,E1 -1815.452,E2 -1815.452} C_VEL
LIN {X 0,Y 580.308,Z 376.827,A -85,B 0,C 180,E1 -1817.624,E2 -1817.624} C_VEL
LIN {X 0,Y 580.307,Z 376.826,A -85,B 0,C 180,E1 -1819.822,E2 -1819.822} C_VEL
LIN {X 0,Y 580.299,Z 376.831,A -85,B 0,C 180,E1 -1822.802,E2 -1822.802} C_VEL
LIN {X 0,Y 580.308,Z 376.827,A -85,B 0,C 180,E1 -1825.08,E2 -1825.08} C_VEL
LIN {X 0,Y 580.304,Z 376.826,A -85,B 0,C 180,E1 -1828.185,E2 -1828.185} C_VEL
LIN {X 0,Y 580.286,Z 376.828,A -85,B 0,C 180,E1 -1830.694,E2 -1830.694} C_VEL
LIN {X 0,Y 580.308,Z 376.825,A -85,B 0,C 180,E1 -1833.316,E2 -1833.316} C_VEL
LIN {X 0,Y 580.248,Z 376.833,A -85,B 0,C 180,E1 -1835.756,E2 -1835.756} C_VEL
LIN {X 0,Y 580.292,Z 376.828,A -85,B 0,C 180,E1 -1838.146,E2 -1838.146} C_VEL
LIN {X 0,Y 580.301,Z 376.826,A -85,B 0,C 180,E1 -1840.843,E2 -1840.843} C_VEL
LIN {X 0,Y 580.292,Z 376.828,A -85,B 0,C 180,E1 -1843.657,E2 -1843.657} C_VEL
LIN {X 0,Y 580.278,Z 376.833,A -85,B 0,C 180,E1 -1846.609,E2 -1846.609} C_VEL
LIN {X 0,Y 580.301,Z 376.829,A -85,B 0,C 180,E1 -1849.156,E2 -1849.156} C_VEL
LIN {X 0,Y 580.332,Z 376.861,A -85,B 0,C 180,E1 -1851.691,E2 -1851.691} C_VEL
LIN {X 0,Y 580.578,Z 382.265,A -85,B 0,C 180,E1 -1852.752,E2 -1852.752} C_VEL
LIN {X 0,Y 580.406,Z 396.664,A -85,B 0,C 180,E1 -1855.426,E2 -1855.426} C_VEL
LIN {X 0,Y 580.761,Z 412.597,A -85,B 0,C 180,E1 -1858.276,E2 -1858.276} C_VEL
LIN {X 0,Y 581,Z 426.983,A -85,B 0,C 180,E1 -1860.817,E2 -1860.817} C_VEL
LIN {X 0,Y 580.83,Z 440.521,A -85,B 0,C 180,E1 -1863.559,E2 -1863.559} C_VEL
LIN {X 0,Y 580.713,Z 453.139,A -85,B 0,C 180,E1 -1866.081,E2 -1866.081} C_VEL
LIN {X 0,Y 580.567,Z 466.848,A -85,B 0,C 180,E1 -1868.767,E2 -1868.767} C_VEL
LIN {X 0,Y 580.475,Z 479.914,A -85,B 0,C 180,E1 -1871.285,E2 -1871.285} C_VEL
LIN {X 0,Y 580.332,Z 495.214,A -85,B 0,C 180,E1 -1874.187,E2 -1874.187} C_VEL
LIN {X 0,Y 580.326,Z 499.881,A -85,B 0,C 180,E1 -1875.053,E2 -1875.053} C_VEL
LIN {X 0,Y 581.151,Z 505.582,A -85,B 0,C 180,E1 -1875.153,E2 -1875.153} C_VEL
LIN {X 0,Y 581.062,Z 520.153,A -85,B 0,C 180,E1 -1875.441,E2 -1875.441} C_VEL
LIN {X 0,Y 580.987,Z 534.578,A -85,B 0,C 180,E1 -1875.88,E2 -1875.88} C_VEL
LIN {X 0,Y 580.856,Z 548.081,A -85,B 0,C 180,E1 -1876.442,E2 -1876.442} C_VEL
LIN {X 0,Y 580.693,Z 561.251,A -85,B 0,C 180,E1 -1877.15,E2 -1877.15} C_VEL
LIN {X 0,Y 580.591,Z 573.137,A -85,B 0,C 180,E1 -1877.947,E2 -1877.947} C_VEL
LIN {X 0,Y 580.443,Z 583.985,A -85,B 0,C 180,E1 -1878.829,E2 -1878.829} C_VEL
LIN {X 0,Y 580.324,Z 594.701,A -85,B 0,C 180,E1 -1879.886,E2 -1879.886} C_VEL
LIN {X 0,Y 580.277,Z 603.554,A -85,B 0,C 180,E1 -1880.94,E2 -1880.94} C_VEL
LIN {X 0,Y 580.199,Z 612.034,A -85,B 0,C 180,E1 -1882.167,E2 -1882.167} C_VEL
LIN {X 0,Y 580.123,Z 618.992,A -85,B 0,C 180,E1 -1883.416,E2 -1883.416} C_VEL
LIN {X 0,Y 580.128,Z 623.565,A -85,B 0,C 180,E1 -1884.438,E2 -1884.438} C_VEL
LIN {X 0,Y 580.102,Z 628.441,A -85,B 0,C 180,E1 -1885.831,E2 -1885.831} C_VEL
LIN {X 0,Y 580.041,Z 631.831,A -85,B 0,C 180,E1 -1887.221,E2 -1887.221} C_VEL
LIN {X 0,Y 580.041,Z 633.831,A -85,B 0,C 180,E1 -1888.611,E2 -1888.611} C_VEL
LIN {X 0,Y 580.036,Z 634.5,A -85,B 0,C 180,E1 -1889.999,E2 -1889.999} C_VEL
LIN {X 0,Y 580.041,Z 633.833,A -85,B 0,C 180,E1 -1891.388,E2 -1891.388} C_VEL
LIN {X 0,Y 580.041,Z 631.833,A -85,B 0,C 180,E1 -1892.777,E2 -1892.777} C_VEL
LIN {X 0,Y 580.102,Z 628.445,A -85,B 0,C 180,E1 -1894.168,E2 -1894.168} C_VEL
LIN {X 0,Y 580.128,Z 623.572,A -85,B 0,C 180,E1 -1895.561,E2 -1895.561} C_VEL
LIN {X 0,Y 580.14,Z 617.057,A -85,B 0,C 180,E1 -1896.957,E2 -1896.957} C_VEL
LIN {X 0,Y 580.191,Z 609.805,A -85,B 0,C 180,E1 -1898.182,E2 -1898.182} C_VEL
LIN {X 0,Y 580.286,Z 600.83,A -85,B 0,C 180,E1 -1899.409,E2 -1899.409} C_VEL
LIN {X 0,Y 580.356,Z 591.4,A -85,B 0,C 180,E1 -1900.465,E2 -1900.465} C_VEL
LIN {X 0,Y 580.474,Z 581.329,A -85,B 0,C 180,E1 -1901.403,E2 -1901.403} C_VEL
LIN {X 0,Y 580.592,Z 569.443,A -85,B 0,C 180,E1 -1902.318,E2 -1902.318} C_VEL
LIN {X 0,Y 580.728,Z 556.663,A -85,B 0,C 180,E1 -1903.114,E2 -1903.114} C_VEL
LIN {X 0,Y 580.874,Z 544.181,A -85,B 0,C 180,E1 -1903.735,E2 -1903.735} C_VEL
LIN {X 0,Y 581.001,Z 531.266,A -85,B 0,C 180,E1 -1904.234,E2 -1904.234} C_VEL
LIN {X 0,Y 581.08,Z 517.23,A -85,B 0,C 180,E1 -1904.63,E2 -1904.63} C_VEL
LIN {X 0,Y 581.089,Z 503.995,A -85,B 0,C 180,E1 -1904.872,E2 -1904.872} C_VEL
LIN {X 0,Y 580.31,Z 499.764,A -85,B 0,C 180,E1 -1904.957,E2 -1904.957} C_VEL
LIN {X 0,Y 580.422,Z 485.66,A -85,B 0,C 180,E1 -1907.62,E2 -1907.62} C_VEL
LIN {X 0,Y 580.509,Z 472.272,A -85,B 0,C 180,E1 -1910.183,E2 -1910.183} C_VEL
LIN {X 0,Y 580.683,Z 456.442,A -85,B 0,C 180,E1 -1913.266,E2 -1913.266} C_VEL
LIN {X 0,Y 580.817,Z 442.03,A -85,B 0,C 180,E1 -1916.136,E2 -1916.136} C_VEL
LIN {X 0,Y 581.012,Z 426.989,A -85,B 0,C 180,E1 -1919.184,E2 -1919.184} C_VEL
LIN {X 0,Y 580.979,Z 411.873,A -85,B 0,C 180,E1 -1922.157,E2 -1922.157} C_VEL
LIN {X 0,Y 581.027,Z 397.748,A -85,B 0,C 180,E1 -1925.066,E2 -1925.066} C_VEL
LIN {X 0,Y 581.253,Z 383.686,A -85,B 0,C 180,E1 -1928.07,E2 -1928.07} C_VEL
LIN {X 0,Y 580.873,Z 379.647,A -85,B 0,C 180,E1 -1928.986,E2 -1928.986} C_VEL
LIN {X 0,Y 580.317,Z 376.827,A -85,B 0,C 180,E1 -1929.687,E2 -1929.687} C_VEL
LIN {X 0,Y 580.275,Z 376.824,A -85,B 0,C 180,E1 -1932.705,E2 -1932.705} C_VEL
LIN {X 0,Y 580.267,Z 376.832,A -85,B 0,C 180,E1 -1935.608,E2 -1935.608} C_VEL
LIN {X 0,Y 580.313,Z 376.822,A -85,B 0,C 180,E1 -1938.234,E2 -1938.234} C_VEL
LIN {X 0,Y 580.283,Z 376.823,A -85,B 0,C 180,E1 -1940.965,E2 -1940.965} C_VEL
LIN {X 0,Y 580.289,Z 376.829,A -85,B 0,C 180,E1 -1943.598,E2 -1943.598} C_VEL
LIN {X 0,Y 580.312,Z 376.822,A -85,B 0,C 180,E1 -1946.145,E2 -1946.145} C_VEL
LIN {X 0,Y 580.283,Z 376.822,A -85,B 0,C 180,E1 -1948.615,E2 -1948.615} C_VEL
LIN {X 0,Y 580.288,Z 376.823,A -85,B 0,C 180,E1 -1951.024,E2 -1951.024} C_VEL
LIN {X 0,Y 580.319,Z 376.827,A -85,B 0,C 180,E1 -1953.658,E2 -1953.658} C_VEL
LIN {X 0,Y 580.271,Z 376.824,A -85,B 0,C 180,E1 -1956.442,E2 -1956.442} C_VEL
LIN {X 0,Y 580.275,Z 376.83,A -85,B 0,C 180,E1 -1959.437,E2 -1959.437} C_VEL
LIN {X 0,Y 580.274,Z 376.832,A -85,B 0,C 180,E1 -1961.645,E2 -1961.645} C_VEL
LIN {X 0,Y 580.276,Z 376.829,A -85,B 0,C 180,E1 -1963.826,E2 -1963.826} C_VEL
LIN {X 0,Y 580.316,Z 376.822,A -85,B 0,C 180,E1 -1965.983,E2 -1965.983} C_VEL
LIN {X 0,Y 580.321,Z 376.818,A -85,B 0,C 180,E1 -1968.827,E2 -1968.827} C_VEL
LIN {X 0,Y 580.326,Z 376.825,A -85,B 0,C 180,E1 -1971.644,E2 -1971.644} C_VEL
LIN {X 0,Y 580.318,Z 376.818,A -85,B 0,C 180,E1 -1974.44,E2 -1974.44} C_VEL
LIN {X 0,Y 580.34,Z 376.821,A -85,B 0,C 180,E1 -1977.224,E2 -1977.224} C_VEL
LIN {X 0,Y 580.342,Z 376.817,A -85,B 0,C 180,E1 -1980,E2 -1980} C_VEL
LIN {X 0,Y 580.339,Z 376.816,A -85,B 0,C 180,E1 -1982.777,E2 -1982.777} C_VEL
LIN {X 0,Y 580.319,Z 376.826,A -85,B 0,C 180,E1 -1985.56,E2 -1985.56} C_VEL
LIN {X 0,Y 580.327,Z 376.817,A -85,B 0,C 180,E1 -1988.356,E2 -1988.356} C_VEL
LIN {X 0,Y 580.323,Z 376.824,A -85,B 0,C 180,E1 -1991.209,E2 -1991.209} C_VEL
LIN {X 0,Y 580.305,Z 376.819,A -85,B 0,C 180,E1 -1994.34,E2 -1994.34} C_VEL
LIN {X 0,Y 580.307,Z 376.823,A -85,B 0,C 180,E1 -1996.916,E2 -1996.916} C_VEL
LIN {X 0,Y 580.3,Z 376.823,A -85,B 0,C 180,E1 -1999.823,E2 -1999.823} C_VEL
LIN {X 0,Y 580.28,Z 376.831,A -85,B 0,C 180,E1 -2001.344,E2 -2001.344} C_VEL
LIN {X 0,Y 579.582,Z 376.912,A -85,B 0,C 180,E1 -2001.924,E2 -2001.924} C_VEL
LIN {X 0,Y 576.704,Z 377.271,A -85,B 0,C 180,E1 -2002.863,E2 -2002.863} C_VEL
LIN {X 0,Y 574.308,Z 377.571,A -85,B 0,C 180,E1 -2003.62,E2 -2003.62} C_VEL
LIN {X 0,Y 573.309,Z 377.691,A -85,B 0,C 180,E1 -2004.204,E2 -2004.204} C_VEL
LIN {X 0,Y 573.243,Z 377.699,A -85,B 0,C 180,E1 -2004.401,E2 -2004.401} C_VEL
LIN {X 0,Y 573.26,Z 377.702,A -85,B 0,C 180,E1 -2006.976,E2 -2006.976} C_VEL
LIN {X 0,Y 573.241,Z 377.706,A -85,B 0,C 180,E1 -2009.49,E2 -2009.49} C_VEL
LIN {X 0,Y 573.25,Z 377.698,A -85,B 0,C 180,E1 -2012.23,E2 -2012.23} C_VEL
LIN {X 0,Y 573.244,Z 377.702,A -85,B 0,C 180,E1 -2014.775,E2 -2014.775} C_VEL
LIN {X 0,Y 573.249,Z 377.708,A -85,B 0,C 180,E1 -2017.167,E2 -2017.167} C_VEL
LIN {X 0,Y 573.243,Z 377.703,A -85,B 0,C 180,E1 -2019.608,E2 -2019.608} C_VEL
LIN {X 0,Y 573.246,Z 377.701,A -85,B 0,C 180,E1 -2022.644,E2 -2022.644} C_VEL
LIN {X 0,Y 573.235,Z 377.703,A -85,B 0,C 180,E1 -2025.668,E2 -2025.668} C_VEL
LIN {X 0,Y 573.241,Z 377.702,A -85,B 0,C 180,E1 -2028.545,E2 -2028.545} C_VEL
LIN {X 0,Y 573.248,Z 377.706,A -85,B 0,C 180,E1 -2031.3,E2 -2031.3} C_VEL
LIN {X 0,Y 573.263,Z 377.697,A -85,B 0,C 180,E1 -2034.012,E2 -2034.012} C_VEL
LIN {X 0,Y 573.284,Z 377.696,A -85,B 0,C 180,E1 -2036.52,E2 -2036.52} C_VEL
LIN {X 0,Y 573.238,Z 377.708,A -85,B 0,C 180,E1 -2039.117,E2 -2039.117} C_VEL
LIN {X 0,Y 573.251,Z 377.698,A -85,B 0,C 180,E1 -2041.972,E2 -2041.972} C_VEL
LIN {X 0,Y 573.256,Z 377.701,A -85,B 0,C 180,E1 -2044.591,E2 -2044.591} C_VEL
LIN {X 0,Y 573.237,Z 377.701,A -85,B 0,C 180,E1 -2047.663,E2 -2047.663} C_VEL
LIN {X 0,Y 573.268,Z 377.702,A -85,B 0,C 180,E1 -2050.671,E2 -2050.671} C_VEL
LIN {X 0,Y 573.245,Z 377.7,A -85,B 0,C 180,E1 -2053.623,E2 -2053.623} C_VEL
LIN {X 0,Y 573.136,Z 377.719,A -85,B 0,C 180,E1 -2055.805,E2 -2055.805} C_VEL
LIN {X 0,Y 573.012,Z 377.735,A -85,B 0,C 180,E1 -2057.247,E2 -2057.247} C_VEL
LIN {X 0,Y 572.978,Z 379.082,A -85,B 0,C 180,E1 -2058.683,E2 -2058.683} C_VEL
LIN {X 0,Y 572.975,Z 381.565,A -85,B 0,C 180,E1 -2060.603,E2 -2060.603} C_VEL
LIN {X 0,Y 573.798,Z 387.594,A -85,B 0,C 180,E1 -2060.75,E2 -2060.75} C_VEL
LIN {X 0,Y 573.758,Z 400.933,A -85,B 0,C 180,E1 -2061.149,E2 -2061.149} C_VEL
LIN {X 0,Y 573.658,Z 412.565,A -85,B 0,C 180,E1 -2061.636,E2 -2061.636} C_VEL
LIN {X 0,Y 573.536,Z 423.951,A -85,B 0,C 180,E1 -2062.254,E2 -2062.254} C_VEL
LIN {X 0,Y 573.374,Z 434.272,A -85,B 0,C 180,E1 -2062.96,E2 -2062.96} C_VEL
LIN {X 0,Y 573.234,Z 444.687,A -85,B 0,C 180,E1 -2063.842,E2 -2063.842} C_VEL
LIN {X 0,Y 573.229,Z 453.171,A -85,B 0,C 180,E1 -2064.725,E2 -2064.725} C_VEL
LIN {X 0,Y 573.145,Z 461.443,A -85,B 0,C 180,E1 -2065.782,E2 -2065.782} C_VEL
LIN {X 0,Y 573.103,Z 468.11,A -85,B 0,C 180,E1 -2066.837,E2 -2066.837} C_VEL
LIN {X 0,Y 572.977,Z 473.443,A -85,B 0,C 180,E1 -2067.892,E2 -2067.892} C_VEL
LIN {X 0,Y 573.01,Z 477.607,A -85,B 0,C 180,E1 -2068.947,E2 -2068.947} C_VEL
LIN {X 0,Y 572.942,Z 480.728,A -85,B 0,C 180,E1 -2070.001,E2 -2070.001} C_VEL
LIN {X 0,Y 572.941,Z 482.28,A -85,B 0,C 180,E1 -2070.704,E2 -2070.704} C_VEL
LIN {X 0,Y 572.948,Z 483.422,A -85,B 0,C 180,E1 -2071.407,E2 -2071.407} C_VEL
LIN {X 0,Y 572.955,Z 484.455,A -85,B 0,C 180,E1 -2072.813,E2 -2072.813} C_VEL
LIN {X 0,Y 573.006,Z 484.401,A -85,B 0,C 180,E1 -2073.517,E2 -2073.517} C_VEL
LIN {X 0,Y 573.008,Z 483.939,A -85,B 0,C 180,E1 -2074.221,E2 -2074.221} C_VEL
LIN {X 0,Y 573.021,Z 481.782,A -85,B 0,C 180,E1 -2075.632,E2 -2075.632} C_VEL
LIN {X 0,Y 573.012,Z 479.491,A -85,B 0,C 180,E1 -2076.549,E2 -2076.549} C_VEL
LIN {X 0,Y 573.021,Z 475.326,A -85,B 0,C 180,E1 -2077.754,E2 -2077.754} C_VEL
LIN {X 0,Y 573.037,Z 470.452,A -85,B 0,C 180,E1 -2078.819,E2 -2078.819} C_VEL
LIN {X 0,Y 573.118,Z 464.292,A -85,B 0,C 180,E1 -2079.886,E2 -2079.886} C_VEL
LIN {X 0,Y 573.17,Z 457.231,A -85,B 0,C 180,E1 -2080.876,E2 -2080.876} C_VEL
LIN {X 0,Y 573.242,Z 448.693,A -85,B 0,C 180,E1 -2081.851,E2 -2081.851} C_VEL
LIN {X 0,Y 573.311,Z 439.052,A -85,B 0,C 180,E1 -2082.748,E2 -2082.748} C_VEL
LIN {X 0,Y 573.456,Z 428.323,A -85,B 0,C 180,E1 -2083.556,E2 -2083.556} C_VEL
LIN {X 0,Y 573.599,Z 416.458,A -85,B 0,C 180,E1 -2084.26,E2 -2084.26} C_VEL
LIN {X 0,Y 573.707,Z 403.514,A -85,B 0,C 180,E1 -2084.846,E2 -2084.846} C_VEL
LIN {X 0,Y 573.828,Z 390.416,A -85,B 0,C 180,E1 -2085.268,E2 -2085.268} C_VEL
LIN {X 0,Y 573.555,Z 385.05,A -85,B 0,C 180,E1 -2085.403,E2 -2085.403} C_VEL
LIN {X 0,Y 572.977,Z 381.407,A -85,B 0,C 180,E1 -2085.496,E2 -2085.496} C_VEL
LIN {X 0,Y 572.967,Z 377.743,A -85,B 0,C 180,E1 -2088.598,E2 -2088.598} C_VEL
LIN {X 0,Y 573.224,Z 377.705,A -85,B 0,C 180,E1 -2091.581,E2 -2091.581} C_VEL
LIN {X 0,Y 573.281,Z 377.698,A -85,B 0,C 180,E1 -2094.634,E2 -2094.634} C_VEL
